	VAR robtarget Openhole_7590 := [[449.75, -1.74, 181.47], [-0.055755, 0.704905, 0.704682, -0.058508], [0,0,0,0], [9E9, 9E9, 9E9, 9E9, 9E9, 9E9]];
	VAR robtarget Openhole_7591 := [[449.26, -1.74, 181.56], [-0.057443, 0.70477, 0.704818, -0.056849], [0,0,0,0], [9E9, 9E9, 9E9, 9E9, 9E9, 9E9]];
	VAR robtarget Openhole_7592 := [[448.77, -1.75, 181.64], [-0.059082, 0.704634, 0.704954, -0.05514], [0,0,0,0], [9E9, 9E9, 9E9, 9E9, 9E9, 9E9]];
	VAR robtarget Openhole_7593 := [[448.27, -1.79, 181.72], [-0.060634, 0.704502, 0.705091, -0.053352], [0,0,0,0], [9E9, 9E9, 9E9, 9E9, 9E9, 9E9]];
	VAR robtarget Openhole_7594 := [[447.79, -1.85, 181.8], [-0.062089, 0.704376, 0.70523, -0.051487], [0,0,0,0], [9E9, 9E9, 9E9, 9E9, 9E9, 9E9]];
	VAR robtarget Openhole_7595 := [[447.3, -1.93, 181.88], [-0.063491, 0.704251, 0.705366, -0.04958], [0,0,0,0], [9E9, 9E9, 9E9, 9E9, 9E9, 9E9]];
	VAR robtarget Openhole_7596 := [[446.81, -2.01, 181.96], [-0.06485, 0.704127, 0.7055, -0.047642], [0,0,0,0], [9E9, 9E9, 9E9, 9E9, 9E9, 9E9]];
	VAR robtarget Openhole_7597 := [[445.85, -2.22, 182.11], [-0.067419, 0.703885, 0.705757, -0.043664], [0,0,0,0], [9E9, 9E9, 9E9, 9E9, 9E9, 9E9]];
	VAR robtarget Openhole_7598 := [[444.89, -2.47, 182.25], [-0.069835, 0.70365, 0.705998, -0.039588], [0,0,0,0], [9E9, 9E9, 9E9, 9E9, 9E9, 9E9]];
	VAR robtarget Openhole_7599 := [[438.19, -4.32, 183.12], [-0.086059, 0.70185, 0.707026, -0.010661], [0,0,0,0], [9E9, 9E9, 9E9, 9E9, 9E9, 9E9]];
	VAR robtarget Openhole_7600 := [[437.22, -4.54, 183.23], [-0.088535, 0.701542, 0.707076, -0.006642], [0,0,0,0], [9E9, 9E9, 9E9, 9E9, 9E9, 9E9]];
	VAR robtarget Openhole_7601 := [[431.68, -6.99, 183.59], [-0.098515, 0.700211, 0.706817, 0.020229], [0,0,0,0], [9E9, 9E9, 9E9, 9E9, 9E9, 9E9]];
	VAR robtarget Openhole_7602 := [[438.07, -6.03, 182.95], [-0.080786, 0.702477, 0.707092, -0.004576], [0,0,0,0], [9E9, 9E9, 9E9, 9E9, 9E9, 9E9]];
	VAR robtarget Openhole_7603 := [[444.39, -4.68, 182.23], [-0.064164, 0.70419, 0.706446, -0.030557], [0,0,0,0], [9E9, 9E9, 9E9, 9E9, 9E9, 9E9]];
	VAR robtarget Openhole_7604 := [[444.87, -4.57, 182.16], [-0.062897, 0.704304, 0.706356, -0.032569], [0,0,0,0], [9E9, 9E9, 9E9, 9E9, 9E9, 9E9]];
	VAR robtarget Openhole_7605 := [[445.84, -4.38, 182.04], [-0.060271, 0.704533, 0.706162, -0.036531], [0,0,0,0], [9E9, 9E9, 9E9, 9E9, 9E9, 9E9]];
	VAR robtarget Openhole_7606 := [[446.33, -4.29, 181.97], [-0.058903, 0.704649, 0.706059, -0.038474], [0,0,0,0], [9E9, 9E9, 9E9, 9E9, 9E9, 9E9]];
	VAR robtarget Openhole_7607 := [[446.82, -4.21, 181.9], [-0.057499, 0.704765, 0.705952, -0.040392], [0,0,0,0], [9E9, 9E9, 9E9, 9E9, 9E9, 9E9]];
	VAR robtarget Openhole_7608 := [[447.31, -4.15, 181.83], [-0.05605, 0.704882, 0.705842, -0.042275], [0,0,0,0], [9E9, 9E9, 9E9, 9E9, 9E9, 9E9]];
	VAR robtarget Openhole_7609 := [[447.81, -4.1, 181.76], [-0.054542, 0.705, 0.70573, -0.044111], [0,0,0,0], [9E9, 9E9, 9E9, 9E9, 9E9, 9E9]];
	VAR robtarget Openhole_7610 := [[448.3, -4.06, 181.69], [-0.053001, 0.705118, 0.705614, -0.04592], [0,0,0,0], [9E9, 9E9, 9E9, 9E9, 9E9, 9E9]];
	VAR robtarget Openhole_7611 := [[448.79, -4.06, 181.62], [-0.051319, 0.705242, 0.705503, -0.047599], [0,0,0,0], [9E9, 9E9, 9E9, 9E9, 9E9, 9E9]];
	VAR robtarget Openhole_7612 := [[449.78, -4.1, 181.48], [-0.047827, 0.705487, 0.705278, -0.050827], [0,0,0,0], [9E9, 9E9, 9E9, 9E9, 9E9, 9E9]];
	VAR robtarget Openhole_7613 := [[450.77, -4.2, 181.34], [-0.04413, 0.705728, 0.705056, -0.053821], [0,0,0,0], [9E9, 9E9, 9E9, 9E9, 9E9, 9E9]];
	VAR robtarget Openhole_7614 := [[456.16, -5.01, 180.62], [-0.022978, 0.706733, 0.703708, -0.069248], [0,0,0,0], [9E9, 9E9, 9E9, 9E9, 9E9, 9E9]];
	VAR robtarget Openhole_7615 := [[458.63, -5.19, 180.3], [-0.013888, 0.70697, 0.702918, -0.07685], [0,0,0,0], [9E9, 9E9, 9E9, 9E9, 9E9, 9E9]];
	VAR robtarget Openhole_7616 := [[459.13, -5.2, 180.24], [-0.012156, 0.707002, 0.702741, -0.078456], [0,0,0,0], [9E9, 9E9, 9E9, 9E9, 9E9, 9E9]];
	VAR robtarget Openhole_7617 := [[463.09, -5.04, 179.69], [0.000811, 0.707106, 0.701098, -0.091987], [0,0,0,0], [9E9, 9E9, 9E9, 9E9, 9E9, 9E9]];
	VAR robtarget Openhole_7618 := [[464.07, -4.96, 179.55], [0.003898, 0.707096, 0.700634, -0.095458], [0,0,0,0], [9E9, 9E9, 9E9, 9E9, 9E9, 9E9]];
	VAR robtarget Openhole_7619 := [[472.91, -4.06, 178.14], [0.030775, 0.706437, 0.695722, -0.126377], [0,0,0,0], [9E9, 9E9, 9E9, 9E9, 9E9, 9E9]];
	VAR robtarget Openhole_7620 := [[478.35, -3.86, 177.31], [0.048077, 0.705471, 0.692398, -0.143474], [0,0,0,0], [9E9, 9E9, 9E9, 9E9, 9E9, 9E9]];
	VAR robtarget Openhole_7621 := [[478.84, -3.85, 177.23], [0.04969, 0.705359, 0.692091, -0.144947], [0,0,0,0], [9E9, 9E9, 9E9, 9E9, 9E9, 9E9]];
	VAR robtarget Openhole_7622 := [[479.33, -3.86, 177.16], [0.051314, 0.705242, 0.691785, -0.146401], [0,0,0,0], [9E9, 9E9, 9E9, 9E9, 9E9, 9E9]];
	VAR robtarget Openhole_7623 := [[480.82, -3.88, 176.95], [0.056219, 0.704868, 0.690865, -0.150682], [0,0,0,0], [9E9, 9E9, 9E9, 9E9, 9E9, 9E9]];
	VAR robtarget Openhole_7624 := [[474.12, -5.49, 178.31], [0.039466, 0.706005, 0.695882, -0.125489], [0,0,0,0], [9E9, 9E9, 9E9, 9E9, 9E9, 9E9]];
	VAR robtarget Openhole_7625 := [[469.21, -6.03, 179.06], [0.024831, 0.706671, 0.698747, -0.108408], [0,0,0,0], [9E9, 9E9, 9E9, 9E9, 9E9, 9E9]];
	VAR robtarget Openhole_7626 := [[460.88, -7.27, 180.24], [0.000752, 0.707106, 0.702859, -0.077394], [0,0,0,0], [9E9, 9E9, 9E9, 9E9, 9E9, 9E9]];
	VAR robtarget Openhole_7627 := [[457.42, -7.57, 180.65], [-0.010088, 0.707035, 0.704119, -0.064938], [0,0,0,0], [9E9, 9E9, 9E9, 9E9, 9E9, 9E9]];
	VAR robtarget Openhole_7628 := [[455.43, -7.61, 180.87], [-0.016739, 0.706909, 0.704712, -0.058151], [0,0,0,0], [9E9, 9E9, 9E9, 9E9, 9E9, 9E9]];
	VAR robtarget Openhole_7629 := [[452.45, -7.48, 181.2], [-0.027374, 0.706577, 0.705437, -0.048573], [0,0,0,0], [9E9, 9E9, 9E9, 9E9, 9E9, 9E9]];
	VAR robtarget Openhole_7630 := [[448.48, -7.26, 181.64], [-0.041664, 0.705878, 0.706196, -0.035883], [0,0,0,0], [9E9, 9E9, 9E9, 9E9, 9E9, 9E9]];
	VAR robtarget Openhole_7631 := [[447.49, -7.25, 181.75], [-0.045079, 0.705668, 0.706357, -0.032546], [0,0,0,0], [9E9, 9E9, 9E9, 9E9, 9E9, 9E9]];
	VAR robtarget Openhole_7632 := [[446.49, -7.27, 181.86], [-0.048387, 0.705449, 0.706508, -0.029104], [0,0,0,0], [9E9, 9E9, 9E9, 9E9, 9E9, 9E9]];
	VAR robtarget Openhole_7633 := [[445.5, -7.33, 181.97], [-0.051524, 0.705227, 0.706647, -0.025509], [0,0,0,0], [9E9, 9E9, 9E9, 9E9, 9E9, 9E9]];
	VAR robtarget Openhole_7634 := [[444.51, -7.43, 182.08], [-0.054538, 0.705, 0.70677, -0.021812], [0,0,0,0], [9E9, 9E9, 9E9, 9E9, 9E9, 9E9]];
	VAR robtarget Openhole_7635 := [[444.02, -7.49, 182.13], [-0.056012, 0.704885, 0.706826, -0.019937], [0,0,0,0], [9E9, 9E9, 9E9, 9E9, 9E9, 9E9]];
	VAR robtarget Openhole_7636 := [[437.6, -8.31, 182.75], [-0.074742, 0.703146, 0.707092, 0.004613], [0,0,0,0], [9E9, 9E9, 9E9, 9E9, 9E9, 9E9]];
	VAR robtarget Openhole_7637 := [[423.69, -9.33, 183.94], [-0.116174, 0.697498, 0.705016, 0.054336], [0,0,0,0], [9E9, 9E9, 9E9, 9E9, 9E9, 9E9]];
	VAR robtarget Openhole_7638 := [[407.25, -10.08, 185.17], [-0.162185, 0.688256, 0.698806, 0.108027], [0,0,0,0], [9E9, 9E9, 9E9, 9E9, 9E9, 9E9]];
	VAR robtarget Openhole_7639 := [[394.36, -10.64, 185.98], [-0.19429, 0.679891, 0.691824, 0.146217], [0,0,0,0], [9E9, 9E9, 9E9, 9E9, 9E9, 9E9]];
	VAR robtarget Openhole_7640 := [[389.36, -10.64, 186.38], [-0.206348, 0.676329, 0.688912, 0.159374], [0,0,0,0], [9E9, 9E9, 9E9, 9E9, 9E9, 9E9]];
	VAR robtarget Openhole_7641 := [[362.36, -10.64, 186.47], [-0.183051, 0.683002, 0.683002, 0.183051], [0,0,0,0], [9E9, 9E9, 9E9, 9E9, 9E9, 9E9]];
	VAR robtarget Openhole_7642 := [[361.72, -33.92, 173.02], [-0.183051, 0.683002, 0.683002, 0.183051], [0,0,0,0], [9E9, 9E9, 9E9, 9E9, 9E9, 9E9]];
	VAR robtarget Openhole_7643 := [[389.32, -33.92, 172.94], [-0.14, 0.693109, 0.670339, 0.225045], [0,0,0,0], [9E9, 9E9, 9E9, 9E9, 9E9, 9E9]];
	VAR robtarget Openhole_7644 := [[399.12, -33.92, 174.34], [-0.112575, 0.698088, 0.677653, 0.201957], [0,0,0,0], [9E9, 9E9, 9E9, 9E9, 9E9, 9E9]];
	VAR robtarget Openhole_7645 := [[405.51, -35.06, 174.78], [-0.090137, 0.701338, 0.681366, 0.18905], [0,0,0,0], [9E9, 9E9, 9E9, 9E9, 9E9, 9E9]];
	VAR robtarget Openhole_7646 := [[411.91, -35.92, 175.46], [-0.067551, 0.703873, 0.685253, 0.174436], [0,0,0,0], [9E9, 9E9, 9E9, 9E9, 9E9, 9E9]];
	VAR robtarget Openhole_7647 := [[417.84, -36.39, 176.28], [-0.046962, 0.705546, 0.688953, 0.159198], [0,0,0,0], [9E9, 9E9, 9E9, 9E9, 9E9, 9E9]];
	VAR robtarget Openhole_7648 := [[421.78, -36.5, 176.91], [-0.033583, 0.706309, 0.691444, 0.148003], [0,0,0,0], [9E9, 9E9, 9E9, 9E9, 9E9, 9E9]];
	VAR robtarget Openhole_7649 := [[422.28, -36.5, 176.99], [-0.031944, 0.706385, 0.691756, 0.146538], [0,0,0,0], [9E9, 9E9, 9E9, 9E9, 9E9, 9E9]];
	VAR robtarget Openhole_7650 := [[428.18, -36.31, 178.02], [-0.012739, 0.706992, 0.69543, 0.127974], [0,0,0,0], [9E9, 9E9, 9E9, 9E9, 9E9, 9E9]];
	VAR robtarget Openhole_7651 := [[436.05, -35.81, 179.39], [0.01245, 0.706997, 0.69979, 0.101457], [0,0,0,0], [9E9, 9E9, 9E9, 9E9, 9E9, 9E9]];
	VAR robtarget Openhole_7652 := [[437.04, -35.79, 179.56], [0.015763, 0.706931, 0.700256, 0.098191], [0,0,0,0], [9E9, 9E9, 9E9, 9E9, 9E9, 9E9]];
	VAR robtarget Openhole_7653 := [[438.02, -35.8, 179.71], [0.019161, 0.706847, 0.700698, 0.094988], [0,0,0,0], [9E9, 9E9, 9E9, 9E9, 9E9, 9E9]];
	VAR robtarget Openhole_7654 := [[439.01, -35.82, 179.87], [0.022643, 0.706744, 0.701116, 0.091853], [0,0,0,0], [9E9, 9E9, 9E9, 9E9, 9E9, 9E9]];
	VAR robtarget Openhole_7655 := [[440, -35.88, 180.03], [0.026226, 0.70662, 0.701507, 0.088811], [0,0,0,0], [9E9, 9E9, 9E9, 9E9, 9E9, 9E9]];
	VAR robtarget Openhole_7656 := [[440.98, -35.98, 180.18], [0.029904, 0.706474, 0.701874, 0.085865], [0,0,0,0], [9E9, 9E9, 9E9, 9E9, 9E9, 9E9]];
	VAR robtarget Openhole_7657 := [[441.96, -36.1, 180.33], [0.033684, 0.706304, 0.702215, 0.083033], [0,0,0,0], [9E9, 9E9, 9E9, 9E9, 9E9, 9E9]];
	VAR robtarget Openhole_7658 := [[442.94, -36.26, 180.48], [0.037548, 0.706109, 0.702532, 0.080306], [0,0,0,0], [9E9, 9E9, 9E9, 9E9, 9E9, 9E9]];
	VAR robtarget Openhole_7659 := [[443.91, -36.44, 180.63], [0.041484, 0.705889, 0.702827, 0.077676], [0,0,0,0], [9E9, 9E9, 9E9, 9E9, 9E9, 9E9]];
	VAR robtarget Openhole_7660 := [[445.84, -36.87, 180.94], [0.049487, 0.705373, 0.703369, 0.072613], [0,0,0,0], [9E9, 9E9, 9E9, 9E9, 9E9, 9E9]];
	VAR robtarget Openhole_7661 := [[446.31, -37, 181.02], [0.051566, 0.705224, 0.703485, 0.071479], [0,0,0,0], [9E9, 9E9, 9E9, 9E9, 9E9, 9E9]];
	VAR robtarget Openhole_7662 := [[446.78, -37.17, 181.09], [0.053699, 0.705065, 0.703588, 0.070455], [0,0,0,0], [9E9, 9E9, 9E9, 9E9, 9E9, 9E9]];
	VAR robtarget Openhole_7663 := [[447.24, -37.35, 181.17], [0.055869, 0.704896, 0.703682, 0.069514], [0,0,0,0], [9E9, 9E9, 9E9, 9E9, 9E9, 9E9]];
	VAR robtarget Openhole_7664 := [[448.2, -37.57, 181.34], [0.059857, 0.704569, 0.703927, 0.066981], [0,0,0,0], [9E9, 9E9, 9E9, 9E9, 9E9, 9E9]];
	VAR robtarget Openhole_7665 := [[448.69, -37.57, 181.42], [0.061551, 0.704423, 0.704081, 0.065341], [0,0,0,0], [9E9, 9E9, 9E9, 9E9, 9E9, 9E9]];
	VAR robtarget Openhole_7666 := [[449.18, -37.57, 181.51], [0.063199, 0.704277, 0.704236, 0.063655], [0,0,0,0], [9E9, 9E9, 9E9, 9E9, 9E9, 9E9]];
	VAR robtarget Openhole_7667 := [[450.15, -37.36, 181.68], [0.065802, 0.704038, 0.70458, 0.059727], [0,0,0,0], [9E9, 9E9, 9E9, 9E9, 9E9, 9E9]];
	VAR robtarget Openhole_7668 := [[450.62, -37.23, 181.76], [0.066984, 0.703927, 0.70475, 0.057688], [0,0,0,0], [9E9, 9E9, 9E9, 9E9, 9E9, 9E9]];
	VAR robtarget Openhole_7669 := [[451.1, -37.12, 181.85], [0.068226, 0.703808, 0.704911, 0.055684], [0,0,0,0], [9E9, 9E9, 9E9, 9E9, 9E9, 9E9]];
	VAR robtarget Openhole_7670 := [[451.58, -36.98, 181.93], [0.069387, 0.703694, 0.70507, 0.053631], [0,0,0,0], [9E9, 9E9, 9E9, 9E9, 9E9, 9E9]];
	VAR robtarget Openhole_7671 := [[459.65, -34.59, 183.08], [0.088452, 0.701553, 0.706872, 0.018235], [0,0,0,0], [9E9, 9E9, 9E9, 9E9, 9E9, 9E9]];
	VAR robtarget Openhole_7672 := [[460.13, -34.45, 183.14], [0.089592, 0.701408, 0.706922, 0.016165], [0,0,0,0], [9E9, 9E9, 9E9, 9E9, 9E9, 9E9]];
	VAR robtarget Openhole_7673 := [[461.11, -32.96, 183.12], [0.087897, 0.701622, 0.707063, 0.007883], [0,0,0,0], [9E9, 9E9, 9E9, 9E9, 9E9, 9E9]];
	VAR robtarget Openhole_7674 := [[460.14, -33.18, 183.01], [0.085435, 0.701927, 0.707006, 0.011915], [0,0,0,0], [9E9, 9E9, 9E9, 9E9, 9E9, 9E9]];
	VAR robtarget Openhole_7675 := [[453.43, -34.99, 182.17], [0.069075, 0.703725, 0.70593, 0.040779], [0,0,0,0], [9E9, 9E9, 9E9, 9E9, 9E9, 9E9]];
	VAR robtarget Openhole_7676 := [[452.47, -35.23, 182.03], [0.066594, 0.703964, 0.705685, 0.044816], [0,0,0,0], [9E9, 9E9, 9E9, 9E9, 9E9, 9E9]];
	VAR robtarget Openhole_7677 := [[451.98, -35.33, 181.96], [0.065304, 0.704085, 0.705556, 0.046802], [0,0,0,0], [9E9, 9E9, 9E9, 9E9, 9E9, 9E9]];
	VAR robtarget Openhole_7678 := [[451.5, -35.42, 181.88], [0.063974, 0.704207, 0.705424, 0.04876], [0,0,0,0], [9E9, 9E9, 9E9, 9E9, 9E9, 9E9]];
	VAR robtarget Openhole_7679 := [[451.01, -35.49, 181.8], [0.062545, 0.704335, 0.705291, 0.050648], [0,0,0,0], [9E9, 9E9, 9E9, 9E9, 9E9, 9E9]];
	VAR robtarget Openhole_7680 := [[450.52, -35.55, 181.73], [0.06107, 0.704465, 0.705155, 0.052498], [0,0,0,0], [9E9, 9E9, 9E9, 9E9, 9E9, 9E9]];
	VAR robtarget Openhole_7681 := [[450.03, -35.58, 181.65], [0.059515, 0.704598, 0.70502, 0.054283], [0,0,0,0], [9E9, 9E9, 9E9, 9E9, 9E9, 9E9]];
	VAR robtarget Openhole_7682 := [[449.53, -35.6, 181.57], [0.057897, 0.704733, 0.704885, 0.056013], [0,0,0,0], [9E9, 9E9, 9E9, 9E9, 9E9, 9E9]];
	VAR robtarget Openhole_7683 := [[449.04, -35.59, 181.49], [0.056177, 0.704872, 0.704754, 0.05764], [0,0,0,0], [9E9, 9E9, 9E9, 9E9, 9E9, 9E9]];
	VAR robtarget Openhole_7684 := [[448.55, -35.55, 181.41], [0.05438, 0.705013, 0.704626, 0.059182], [0,0,0,0], [9E9, 9E9, 9E9, 9E9, 9E9, 9E9]];
	VAR robtarget Openhole_7685 := [[448.06, -35.5, 181.34], [0.052527, 0.705153, 0.7045, 0.06066], [0,0,0,0], [9E9, 9E9, 9E9, 9E9, 9E9, 9E9]];
	VAR robtarget Openhole_7686 := [[447.57, -35.43, 181.26], [0.050625, 0.705292, 0.704377, 0.062073], [0,0,0,0], [9E9, 9E9, 9E9, 9E9, 9E9, 9E9]];
	VAR robtarget Openhole_7687 := [[446.59, -35.25, 181.11], [0.04671, 0.705562, 0.704136, 0.064752], [0,0,0,0], [9E9, 9E9, 9E9, 9E9, 9E9, 9E9]];
	VAR robtarget Openhole_7688 := [[443.68, -34.65, 180.69], [0.034788, 0.706251, 0.703375, 0.072552], [0,0,0,0], [9E9, 9E9, 9E9, 9E9, 9E9, 9E9]];
	VAR robtarget Openhole_7689 := [[441.73, -34.35, 180.42], [0.027076, 0.706588, 0.702783, 0.078074], [0,0,0,0], [9E9, 9E9, 9E9, 9E9, 9E9, 9E9]];
	VAR robtarget Openhole_7690 := [[440.74, -34.25, 180.28], [0.023353, 0.706721, 0.702453, 0.080994], [0,0,0,0], [9E9, 9E9, 9E9, 9E9, 9E9, 9E9]];
	VAR robtarget Openhole_7691 := [[439.75, -34.17, 180.14], [0.019722, 0.706832, 0.702098, 0.084012], [0,0,0,0], [9E9, 9E9, 9E9, 9E9, 9E9, 9E9]];
	VAR robtarget Openhole_7692 := [[438.76, -34.13, 180], [0.016187, 0.706921, 0.701719, 0.087122], [0,0,0,0], [9E9, 9E9, 9E9, 9E9, 9E9, 9E9]];
	VAR robtarget Openhole_7693 := [[437.77, -34.12, 179.86], [0.012758, 0.706992, 0.701314, 0.090326], [0,0,0,0], [9E9, 9E9, 9E9, 9E9, 9E9, 9E9]];
	VAR robtarget Openhole_7694 := [[437.28, -34.12, 179.79], [0.01108, 0.70702, 0.701102, 0.091956], [0,0,0,0], [9E9, 9E9, 9E9, 9E9, 9E9, 9E9]];
	VAR robtarget Openhole_7695 := [[431.85, -34.44, 178.95], [-0.00638, 0.707078, 0.698424, 0.110474], [0,0,0,0], [9E9, 9E9, 9E9, 9E9, 9E9, 9E9]];
	VAR robtarget Openhole_7696 := [[424.96, -34.89, 177.82], [-0.028192, 0.706545, 0.694415, 0.133373], [0,0,0,0], [9E9, 9E9, 9E9, 9E9, 9E9, 9E9]];
	VAR robtarget Openhole_7697 := [[422, -34.94, 177.35], [-0.037884, 0.706091, 0.692603, 0.142482], [0,0,0,0], [9E9, 9E9, 9E9, 9E9, 9E9, 9E9]];
	VAR robtarget Openhole_7698 := [[421.5, -34.94, 177.28], [-0.039531, 0.706001, 0.6923, 0.143945], [0,0,0,0], [9E9, 9E9, 9E9, 9E9, 9E9, 9E9]];
	VAR robtarget Openhole_7699 := [[415.57, -34.71, 176.45], [-0.059667, 0.704585, 0.688649, 0.160508], [0,0,0,0], [9E9, 9E9, 9E9, 9E9, 9E9, 9E9]];
	VAR robtarget Openhole_7700 := [[409.14, -34.09, 175.71], [-0.081938, 0.702343, 0.684724, 0.176502], [0,0,0,0], [9E9, 9E9, 9E9, 9E9, 9E9, 9E9]];
	VAR robtarget Openhole_7701 := [[404.2, -33.45, 175.28], [-0.099015, 0.70014, 0.681745, 0.187681], [0,0,0,0], [9E9, 9E9, 9E9, 9E9, 9E9, 9E9]];
	VAR robtarget Openhole_7702 := [[411.67, -32.92, 176.51], [-0.077704, 0.702824, 0.687349, 0.165988], [0,0,0,0], [9E9, 9E9, 9E9, 9E9, 9E9, 9E9]];
	VAR robtarget Openhole_7703 := [[418.12, -33.28, 177.26], [-0.055972, 0.704888, 0.691289, 0.148726], [0,0,0,0], [9E9, 9E9, 9E9, 9E9, 9E9, 9E9]];
	VAR robtarget Openhole_7704 := [[420.6, -33.32, 177.59], [-0.047766, 0.705492, 0.692797, 0.141538], [0,0,0,0], [9E9, 9E9, 9E9, 9E9, 9E9, 9E9]];
	VAR robtarget Openhole_7705 := [[421.09, -33.31, 177.66], [-0.046147, 0.705599, 0.693098, 0.140056], [0,0,0,0], [9E9, 9E9, 9E9, 9E9, 9E9, 9E9]];
	VAR robtarget Openhole_7706 := [[426.53, -33.08, 178.46], [-0.028845, 0.706518, 0.696362, 0.122803], [0,0,0,0], [9E9, 9E9, 9E9, 9E9, 9E9, 9E9]];
	VAR robtarget Openhole_7707 := [[436.37, -32.09, 179.91], [0.001199, 0.707106, 0.701578, 0.088254], [0,0,0,0], [9E9, 9E9, 9E9, 9E9, 9E9, 9E9]];
	VAR robtarget Openhole_7708 := [[438.85, -31.99, 180.23], [0.009317, 0.707045, 0.70259, 0.079793], [0,0,0,0], [9E9, 9E9, 9E9, 9E9, 9E9, 9E9]];
	VAR robtarget Openhole_7709 := [[439.84, -31.99, 180.36], [0.012734, 0.706992, 0.702952, 0.07654], [0,0,0,0], [9E9, 9E9, 9E9, 9E9, 9E9, 9E9]];
	VAR robtarget Openhole_7710 := [[441.33, -32.04, 180.54], [0.017999, 0.706878, 0.703454, 0.071779], [0,0,0,0], [9E9, 9E9, 9E9, 9E9, 9E9, 9E9]];
	VAR robtarget Openhole_7711 := [[442.32, -32.11, 180.66], [0.021607, 0.706777, 0.703762, 0.068696], [0,0,0,0], [9E9, 9E9, 9E9, 9E9, 9E9, 9E9]];
	VAR robtarget Openhole_7712 := [[442.81, -32.16, 180.72], [0.023462, 0.706717, 0.703905, 0.06721], [0,0,0,0], [9E9, 9E9, 9E9, 9E9, 9E9, 9E9]];
	VAR robtarget Openhole_7713 := [[447.23, -32.82, 181.26], [0.040783, 0.70593, 0.704996, 0.054591], [0,0,0,0], [9E9, 9E9, 9E9, 9E9, 9E9, 9E9]];
	VAR robtarget Openhole_7714 := [[448.21, -32.96, 181.39], [0.044601, 0.705699, 0.705211, 0.051745], [0,0,0,0], [9E9, 9E9, 9E9, 9E9, 9E9, 9E9]];
	VAR robtarget Openhole_7715 := [[448.7, -33.01, 181.45], [0.046456, 0.705579, 0.705319, 0.050252], [0,0,0,0], [9E9, 9E9, 9E9, 9E9, 9E9, 9E9]];
	VAR robtarget Openhole_7716 := [[449.2, -33.05, 181.52], [0.048263, 0.705458, 0.705427, 0.048706], [0,0,0,0], [9E9, 9E9, 9E9, 9E9, 9E9, 9E9]];
	VAR robtarget Openhole_7717 := [[449.69, -33.07, 181.59], [0.05002, 0.705335, 0.705536, 0.047102], [0,0,0,0], [9E9, 9E9, 9E9, 9E9, 9E9, 9E9]];
	VAR robtarget Openhole_7718 := [[450.19, -33.08, 181.65], [0.051725, 0.705212, 0.705645, 0.045443], [0,0,0,0], [9E9, 9E9, 9E9, 9E9, 9E9, 9E9]];
	VAR robtarget Openhole_7719 := [[451.18, -33.03, 181.79], [0.054938, 0.704969, 0.705862, 0.041938], [0,0,0,0], [9E9, 9E9, 9E9, 9E9, 9E9, 9E9]];
	VAR robtarget Openhole_7720 := [[451.67, -32.99, 181.85], [0.056457, 0.704849, 0.705968, 0.04011], [0,0,0,0], [9E9, 9E9, 9E9, 9E9, 9E9, 9E9]];
	VAR robtarget Openhole_7721 := [[452.16, -32.92, 181.92], [0.057903, 0.704732, 0.706073, 0.038223], [0,0,0,0], [9E9, 9E9, 9E9, 9E9, 9E9, 9E9]];
	VAR robtarget Openhole_7722 := [[452.65, -32.84, 181.98], [0.059299, 0.704616, 0.706174, 0.036299], [0,0,0,0], [9E9, 9E9, 9E9, 9E9, 9E9, 9E9]];
	VAR robtarget Openhole_7723 := [[453.63, -32.66, 182.1], [0.061962, 0.704387, 0.706366, 0.032359], [0,0,0,0], [9E9, 9E9, 9E9, 9E9, 9E9, 9E9]];
	VAR robtarget Openhole_7724 := [[460.44, -31.22, 182.84], [0.07991, 0.702577, 0.707093, 0.004382], [0,0,0,0], [9E9, 9E9, 9E9, 9E9, 9E9, 9E9]];
	VAR robtarget Openhole_7725 := [[466.84, -30.31, 183.44], [0.097818, 0.700308, 0.706815, -0.020309], [0,0,0,0], [9E9, 9E9, 9E9, 9E9, 9E9, 9E9]];
	VAR robtarget Openhole_7726 := [[476.26, -29.36, 184.22], [0.12433, 0.69609, 0.704993, -0.054634], [0,0,0,0], [9E9, 9E9, 9E9, 9E9, 9E9, 9E9]];
	VAR robtarget Openhole_7727 := [[470.3, -26.56, 183.06], [0.096566, 0.700482, 0.705722, -0.044238], [0,0,0,0], [9E9, 9E9, 9E9, 9E9, 9E9, 9E9]];
	VAR robtarget Openhole_7728 := [[465.31, -26.64, 182.71], [0.080722, 0.702484, 0.706578, -0.027351], [0,0,0,0], [9E9, 9E9, 9E9, 9E9, 9E9, 9E9]];
	VAR robtarget Openhole_7729 := [[464.82, -26.64, 182.67], [0.079088, 0.70267, 0.70664, -0.025682], [0,0,0,0], [9E9, 9E9, 9E9, 9E9, 9E9, 9E9]];
	VAR robtarget Openhole_7730 := [[463.82, -26.63, 182.6], [0.075801, 0.703032, 0.706754, -0.022343], [0,0,0,0], [9E9, 9E9, 9E9, 9E9, 9E9, 9E9]];
	VAR robtarget Openhole_7731 := [[463.32, -26.64, 182.56], [0.074164, 0.703207, 0.706805, -0.020661], [0,0,0,0], [9E9, 9E9, 9E9, 9E9, 9E9, 9E9]];
	VAR robtarget Openhole_7732 := [[462.82, -26.63, 182.53], [0.072502, 0.70338, 0.706852, -0.018998], [0,0,0,0], [9E9, 9E9, 9E9, 9E9, 9E9, 9E9]];
	VAR robtarget Openhole_7733 := [[459.33, -26.59, 182.27], [0.060784, 0.704489, 0.707069, -0.007327], [0,0,0,0], [9E9, 9E9, 9E9, 9E9, 9E9, 9E9]];
	VAR robtarget Openhole_7734 := [[458.83, -26.59, 182.23], [0.059117, 0.704631, 0.707084, -0.005637], [0,0,0,0], [9E9, 9E9, 9E9, 9E9, 9E9, 9E9]];
	VAR robtarget Openhole_7735 := [[458.33, -26.6, 182.2], [0.057459, 0.704768, 0.707096, -0.003935], [0,0,0,0], [9E9, 9E9, 9E9, 9E9, 9E9, 9E9]];
	VAR robtarget Openhole_7736 := [[457.83, -26.59, 182.16], [0.055777, 0.704903, 0.707103, -0.002253], [0,0,0,0], [9E9, 9E9, 9E9, 9E9, 9E9, 9E9]];
	VAR robtarget Openhole_7737 := [[456.34, -26.58, 182.05], [0.050691, 0.705287, 0.707101, 0.002767], [0,0,0,0], [9E9, 9E9, 9E9, 9E9, 9E9, 9E9]];
	VAR robtarget Openhole_7738 := [[455.34, -26.54, 181.97], [0.04721, 0.705529, 0.707081, 0.006033], [0,0,0,0], [9E9, 9E9, 9E9, 9E9, 9E9, 9E9]];
	VAR robtarget Openhole_7739 := [[454.85, -26.49, 181.94], [0.045376, 0.705649, 0.707066, 0.007562], [0,0,0,0], [9E9, 9E9, 9E9, 9E9, 9E9, 9E9]];
	VAR robtarget Openhole_7740 := [[454.35, -26.44, 181.9], [0.043506, 0.705767, 0.707049, 0.009049], [0,0,0,0], [9E9, 9E9, 9E9, 9E9, 9E9, 9E9]];
	VAR robtarget Openhole_7741 := [[453.86, -26.35, 181.86], [0.041562, 0.705884, 0.70703, 0.01044], [0,0,0,0], [9E9, 9E9, 9E9, 9E9, 9E9, 9E9]];
	VAR robtarget Openhole_7742 := [[453.37, -26.25, 181.82], [0.03957, 0.705999, 0.707009, 0.011766], [0,0,0,0], [9E9, 9E9, 9E9, 9E9, 9E9, 9E9]];
	VAR robtarget Openhole_7743 := [[452.79, -25.92, 181.77], [0.036472, 0.706166, 0.706994, 0.012621], [0,0,0,0], [9E9, 9E9, 9E9, 9E9, 9E9, 9E9]];
	VAR robtarget Openhole_7744 := [[454.94, -24.42, 181.83], [0.038676, 0.706048, 0.707107, 0.000228], [0,0,0,0], [9E9, 9E9, 9E9, 9E9, 9E9, 9E9]];
	VAR robtarget Openhole_7745 := [[455.54, -24.57, 181.87], [0.041225, 0.705904, 0.707106, -0.001297], [0,0,0,0], [9E9, 9E9, 9E9, 9E9, 9E9, 9E9]];
	VAR robtarget Openhole_7746 := [[456.54, -24.66, 181.93], [0.044874, 0.705681, 0.707093, -0.004383], [0,0,0,0], [9E9, 9E9, 9E9, 9E9, 9E9, 9E9]];
	VAR robtarget Openhole_7747 := [[457.04, -24.68, 181.96], [0.046645, 0.705567, 0.707081, -0.005982], [0,0,0,0], [9E9, 9E9, 9E9, 9E9, 9E9, 9E9]];
	VAR robtarget Openhole_7748 := [[460.52, -24.98, 182.18], [0.059311, 0.704615, 0.706908, -0.016769], [0,0,0,0], [9E9, 9E9, 9E9, 9E9, 9E9, 9E9]];
	VAR robtarget Openhole_7749 := [[457.19, -28.45, 182.25], [0.059837, 0.70457, 0.70708, 0.006176], [0,0,0,0], [9E9, 9E9, 9E9, 9E9, 9E9, 9E9]];
	VAR robtarget Openhole_7750 := [[454.2, -28.65, 181.99], [0.050478, 0.705303, 0.706903, 0.01699], [0,0,0,0], [9E9, 9E9, 9E9, 9E9, 9E9, 9E9]];
	VAR robtarget Openhole_7751 := [[453.71, -28.66, 181.95], [0.048836, 0.705418, 0.706859, 0.018724], [0,0,0,0], [9E9, 9E9, 9E9, 9E9, 9E9, 9E9]];
	VAR robtarget Openhole_7752 := [[452.71, -28.67, 181.85], [0.045488, 0.705642, 0.70676, 0.022133], [0,0,0,0], [9E9, 9E9, 9E9, 9E9, 9E9, 9E9]];
	VAR robtarget Openhole_7753 := [[449.23, -28.52, 181.53], [0.033165, 0.706329, 0.706314, 0.033467], [0,0,0,0], [9E9, 9E9, 9E9, 9E9, 9E9, 9E9]];
	VAR robtarget Openhole_7754 := [[448.73, -28.52, 181.49], [0.031442, 0.706407, 0.706234, 0.035127], [0,0,0,0], [9E9, 9E9, 9E9, 9E9, 9E9, 9E9]];
	VAR robtarget Openhole_7755 := [[448.23, -28.52, 181.44], [0.029744, 0.706481, 0.706148, 0.036814], [0,0,0,0], [9E9, 9E9, 9E9, 9E9, 9E9, 9E9]];
	VAR robtarget Openhole_7756 := [[447.24, -28.52, 181.35], [0.026357, 0.706615, 0.705964, 0.040193], [0,0,0,0], [9E9, 9E9, 9E9, 9E9, 9E9, 9E9]];
	VAR robtarget Openhole_7757 := [[444.75, -28.61, 181.12], [0.01815, 0.706874, 0.705416, 0.048872], [0,0,0,0], [9E9, 9E9, 9E9, 9E9, 9E9, 9E9]];
	VAR robtarget Openhole_7758 := [[443.26, -28.67, 180.98], [0.013272, 0.706982, 0.705034, 0.054102], [0,0,0,0], [9E9, 9E9, 9E9, 9E9, 9E9, 9E9]];
	VAR robtarget Openhole_7759 := [[444.55, -31.6, 180.96], [0.02758, 0.706569, 0.704595, 0.059544], [0,0,0,0], [9E9, 9E9, 9E9, 9E9, 9E9, 9E9]];
	VAR robtarget Openhole_7760 := [[445.54, -31.73, 181.08], [0.03138, 0.70641, 0.704833, 0.056663], [0,0,0,0], [9E9, 9E9, 9E9, 9E9, 9E9, 9E9]];
	VAR robtarget Openhole_7761 := [[446.52, -31.9, 181.19], [0.035276, 0.706226, 0.705049, 0.05391], [0,0,0,0], [9E9, 9E9, 9E9, 9E9, 9E9, 9E9]];
	VAR robtarget Openhole_7762 := [[448.49, -32.14, 181.43], [0.042816, 0.705809, 0.705471, 0.048074], [0,0,0,0], [9E9, 9E9, 9E9, 9E9, 9E9, 9E9]];
	VAR robtarget Openhole_7763 := [[448.98, -32.18, 181.5], [0.044643, 0.705696, 0.705573, 0.046543], [0,0,0,0], [9E9, 9E9, 9E9, 9E9, 9E9, 9E9]];
	VAR robtarget Openhole_7764 := [[449.48, -32.21, 181.56], [0.046426, 0.705581, 0.705676, 0.044962], [0,0,0,0], [9E9, 9E9, 9E9, 9E9, 9E9, 9E9]];
	VAR robtarget Openhole_7765 := [[449.97, -32.23, 181.62], [0.048173, 0.705464, 0.705777, 0.043345], [0,0,0,0], [9E9, 9E9, 9E9, 9E9, 9E9, 9E9]];
	VAR robtarget Openhole_7766 := [[450.47, -32.23, 181.68], [0.049855, 0.705347, 0.705879, 0.041659], [0,0,0,0], [9E9, 9E9, 9E9, 9E9, 9E9, 9E9]];
	VAR robtarget Openhole_7767 := [[450.97, -32.22, 181.75], [0.051492, 0.705229, 0.705978, 0.039931], [0,0,0,0], [9E9, 9E9, 9E9, 9E9, 9E9, 9E9]];
	VAR robtarget Openhole_7768 := [[451.46, -32.18, 181.81], [0.053057, 0.705113, 0.706078, 0.038137], [0,0,0,0], [9E9, 9E9, 9E9, 9E9, 9E9, 9E9]];
	VAR robtarget Openhole_7769 := [[451.96, -32.13, 181.87], [0.054571, 0.704998, 0.706174, 0.036302], [0,0,0,0], [9E9, 9E9, 9E9, 9E9, 9E9, 9E9]];
	VAR robtarget Openhole_7770 := [[452.45, -32.07, 181.93], [0.056024, 0.704884, 0.706269, 0.034416], [0,0,0,0], [9E9, 9E9, 9E9, 9E9, 9E9, 9E9]];
	VAR robtarget Openhole_7771 := [[453.43, -31.9, 182.05], [0.058774, 0.70466, 0.706447, 0.03053], [0,0,0,0], [9E9, 9E9, 9E9, 9E9, 9E9, 9E9]];
	VAR robtarget Openhole_7772 := [[452.74, -30.49, 181.92], [0.051737, 0.705211, 0.706546, 0.028148], [0,0,0,0], [9E9, 9E9, 9E9, 9E9, 9E9, 9E9]];
	VAR robtarget Openhole_7773 := [[451.25, -30.57, 181.75], [0.046945, 0.705547, 0.706315, 0.033461], [0,0,0,0], [9E9, 9E9, 9E9, 9E9, 9E9, 9E9]];
	VAR robtarget Openhole_7774 := [[450.76, -30.57, 181.7], [0.045265, 0.705656, 0.706232, 0.035156], [0,0,0,0], [9E9, 9E9, 9E9, 9E9, 9E9, 9E9]];
	VAR robtarget Openhole_7775 := [[450.26, -30.57, 181.64], [0.043559, 0.705764, 0.706147, 0.036824], [0,0,0,0], [9E9, 9E9, 9E9, 9E9, 9E9, 9E9]];
	VAR robtarget Openhole_7776 := [[446.79, -30.31, 181.26], [0.030887, 0.706432, 0.705495, 0.047722], [0,0,0,0], [9E9, 9E9, 9E9, 9E9, 9E9, 9E9]];

	PROC MainOpenhole()
		moveJ Openhole_0, v10, fine, pHeader\WObj:=wobj0;
		MoveL Openhole_1, v10, fine, pHeader\WObj:=wobj0;
		MoveL Openhole_2, v10, fine, pHeader\WObj:=wobj0;
		MoveL Openhole_3, v10, fine, pHeader\WObj:=wobj0;
		MoveL Openhole_4, v10, fine, pHeader\WObj:=wobj0;
		MoveL Openhole_5, v10, fine, pHeader\WObj:=wobj0;
		MoveL Openhole_6, v10, fine, pHeader\WObj:=wobj0;
		MoveL Openhole_7, v10, fine, pHeader\WObj:=wobj0;
		MoveL Openhole_8, v10, fine, pHeader\WObj:=wobj0;
		MoveL Openhole_9, v10, fine, pHeader\WObj:=wobj0;
		MoveL Openhole_10, v10, fine, pHeader\WObj:=wobj0;
		MoveL Openhole_11, v10, fine, pHeader\WObj:=wobj0;
		MoveL Openhole_12, v10, fine, pHeader\WObj:=wobj0;
		MoveL Openhole_13, v10, fine, pHeader\WObj:=wobj0;
		MoveL Openhole_14, v10, fine, pHeader\WObj:=wobj0;
		MoveL Openhole_15, v10, fine, pHeader\WObj:=wobj0;
		MoveL Openhole_16, v10, fine, pHeader\WObj:=wobj0;
		MoveL Openhole_17, v10, fine, pHeader\WObj:=wobj0;
		MoveL Openhole_18, v10, fine, pHeader\WObj:=wobj0;
		MoveL Openhole_19, v10, fine, pHeader\WObj:=wobj0;
		MoveL Openhole_20, v10, fine, pHeader\WObj:=wobj0;
		MoveL Openhole_21, v10, fine, pHeader\WObj:=wobj0;
		MoveL Openhole_22, v10, fine, pHeader\WObj:=wobj0;
		MoveL Openhole_23, v10, fine, pHeader\WObj:=wobj0;
		MoveL Openhole_24, v10, fine, pHeader\WObj:=wobj0;
		MoveL Openhole_25, v10, fine, pHeader\WObj:=wobj0;
		MoveL Openhole_26, v10, fine, pHeader\WObj:=wobj0;
		MoveL Openhole_27, v10, fine, pHeader\WObj:=wobj0;
		MoveL Openhole_28, v10, fine, pHeader\WObj:=wobj0;
		MoveL Openhole_29, v10, fine, pHeader\WObj:=wobj0;
		MoveL Openhole_30, v10, fine, pHeader\WObj:=wobj0;
		MoveL Openhole_31, v10, fine, pHeader\WObj:=wobj0;
		MoveL Openhole_32, v10, fine, pHeader\WObj:=wobj0;
		MoveL Openhole_33, v10, fine, pHeader\WObj:=wobj0;
		MoveL Openhole_34, v10, fine, pHeader\WObj:=wobj0;
		MoveL Openhole_35, v10, fine, pHeader\WObj:=wobj0;
		MoveL Openhole_36, v10, fine, pHeader\WObj:=wobj0;
		MoveL Openhole_37, v10, fine, pHeader\WObj:=wobj0;
		MoveL Openhole_38, v10, fine, pHeader\WObj:=wobj0;
		MoveL Openhole_39, v10, fine, pHeader\WObj:=wobj0;
		MoveL Openhole_40, v10, fine, pHeader\WObj:=wobj0;
		MoveL Openhole_41, v10, fine, pHeader\WObj:=wobj0;
		MoveL Openhole_42, v10, fine, pHeader\WObj:=wobj0;
		MoveL Openhole_43, v10, fine, pHeader\WObj:=wobj0;
		MoveL Openhole_44, v10, fine, pHeader\WObj:=wobj0;
		MoveL Openhole_45, v10, fine, pHeader\WObj:=wobj0;
		MoveL Openhole_46, v10, fine, pHeader\WObj:=wobj0;
		MoveL Openhole_47, v10, fine, pHeader\WObj:=wobj0;
		MoveL Openhole_48, v10, fine, pHeader\WObj:=wobj0;
		MoveL Openhole_49, v10, fine, pHeader\WObj:=wobj0;
		MoveL Openhole_50, v10, fine, pHeader\WObj:=wobj0;
		MoveL Openhole_51, v10, fine, pHeader\WObj:=wobj0;
		MoveL Openhole_52, v10, fine, pHeader\WObj:=wobj0;
		MoveL Openhole_53, v10, fine, pHeader\WObj:=wobj0;
		MoveL Openhole_54, v10, fine, pHeader\WObj:=wobj0;
		MoveL Openhole_55, v10, fine, pHeader\WObj:=wobj0;
		MoveL Openhole_56, v10, fine, pHeader\WObj:=wobj0;
		MoveL Openhole_57, v10, fine, pHeader\WObj:=wobj0;
		MoveL Openhole_58, v10, fine, pHeader\WObj:=wobj0;
		MoveL Openhole_59, v10, fine, pHeader\WObj:=wobj0;
		MoveL Openhole_60, v10, fine, pHeader\WObj:=wobj0;
		MoveL Openhole_61, v10, fine, pHeader\WObj:=wobj0;
		MoveL Openhole_62, v10, fine, pHeader\WObj:=wobj0;
		MoveL Openhole_63, v10, fine, pHeader\WObj:=wobj0;
		MoveL Openhole_64, v10, fine, pHeader\WObj:=wobj0;
		MoveL Openhole_65, v10, fine, pHeader\WObj:=wobj0;
		MoveL Openhole_66, v10, fine, pHeader\WObj:=wobj0;
		MoveL Openhole_67, v10, fine, pHeader\WObj:=wobj0;
		MoveL Openhole_68, v10, fine, pHeader\WObj:=wobj0;
		MoveL Openhole_69, v10, fine, pHeader\WObj:=wobj0;
		MoveL Openhole_70, v10, fine, pHeader\WObj:=wobj0;
		MoveL Openhole_71, v10, fine, pHeader\WObj:=wobj0;
		MoveL Openhole_72, v10, fine, pHeader\WObj:=wobj0;
		MoveL Openhole_73, v10, fine, pHeader\WObj:=wobj0;
		MoveL Openhole_74, v10, fine, pHeader\WObj:=wobj0;
		MoveL Openhole_75, v10, fine, pHeader\WObj:=wobj0;
		MoveL Openhole_76, v10, fine, pHeader\WObj:=wobj0;
		MoveL Openhole_77, v10, fine, pHeader\WObj:=wobj0;
		MoveL Openhole_78, v10, fine, pHeader\WObj:=wobj0;
		MoveL Openhole_79, v10, fine, pHeader\WObj:=wobj0;
		MoveL Openhole_80, v10, fine, pHeader\WObj:=wobj0;
		MoveL Openhole_81, v10, fine, pHeader\WObj:=wobj0;
		MoveL Openhole_82, v10, fine, pHeader\WObj:=wobj0;
		MoveL Openhole_83, v10, fine, pHeader\WObj:=wobj0;
		MoveL Openhole_84, v10, fine, pHeader\WObj:=wobj0;
		MoveL Openhole_85, v10, fine, pHeader\WObj:=wobj0;
		MoveL Openhole_86, v10, fine, pHeader\WObj:=wobj0;
		MoveL Openhole_87, v10, fine, pHeader\WObj:=wobj0;
		MoveL Openhole_88, v10, fine, pHeader\WObj:=wobj0;
		MoveL Openhole_89, v10, fine, pHeader\WObj:=wobj0;
		MoveL Openhole_90, v10, fine, pHeader\WObj:=wobj0;
		MoveL Openhole_91, v10, fine, pHeader\WObj:=wobj0;
		MoveL Openhole_92, v10, fine, pHeader\WObj:=wobj0;
		MoveL Openhole_93, v10, fine, pHeader\WObj:=wobj0;
		MoveL Openhole_94, v10, fine, pHeader\WObj:=wobj0;
		MoveL Openhole_95, v10, fine, pHeader\WObj:=wobj0;
		MoveL Openhole_96, v10, fine, pHeader\WObj:=wobj0;
		MoveL Openhole_97, v10, fine, pHeader\WObj:=wobj0;
		MoveL Openhole_98, v10, fine, pHeader\WObj:=wobj0;
		MoveL Openhole_99, v10, fine, pHeader\WObj:=wobj0;
		MoveL Openhole_100, v10, fine, pHeader\WObj:=wobj0;
		MoveL Openhole_101, v10, fine, pHeader\WObj:=wobj0;
		MoveL Openhole_102, v10, fine, pHeader\WObj:=wobj0;
		MoveL Openhole_103, v10, fine, pHeader\WObj:=wobj0;
		MoveL Openhole_104, v10, fine, pHeader\WObj:=wobj0;
		MoveL Openhole_105, v10, fine, pHeader\WObj:=wobj0;
		MoveL Openhole_106, v10, fine, pHeader\WObj:=wobj0;
		MoveL Openhole_107, v10, fine, pHeader\WObj:=wobj0;
		MoveL Openhole_108, v10, fine, pHeader\WObj:=wobj0;
		MoveL Openhole_109, v10, fine, pHeader\WObj:=wobj0;
		MoveL Openhole_110, v10, fine, pHeader\WObj:=wobj0;
		MoveL Openhole_111, v10, fine, pHeader\WObj:=wobj0;
		MoveL Openhole_112, v10, fine, pHeader\WObj:=wobj0;
		MoveL Openhole_113, v10, fine, pHeader\WObj:=wobj0;
		MoveL Openhole_114, v10, fine, pHeader\WObj:=wobj0;
		MoveL Openhole_115, v10, fine, pHeader\WObj:=wobj0;
		MoveL Openhole_116, v10, fine, pHeader\WObj:=wobj0;
		MoveL Openhole_117, v10, fine, pHeader\WObj:=wobj0;
		MoveL Openhole_118, v10, fine, pHeader\WObj:=wobj0;
		MoveL Openhole_119, v10, fine, pHeader\WObj:=wobj0;
		MoveL Openhole_120, v10, fine, pHeader\WObj:=wobj0;
		MoveL Openhole_121, v10, fine, pHeader\WObj:=wobj0;
		MoveL Openhole_122, v10, fine, pHeader\WObj:=wobj0;
		MoveL Openhole_123, v10, fine, pHeader\WObj:=wobj0;
		MoveL Openhole_124, v10, fine, pHeader\WObj:=wobj0;
		MoveL Openhole_125, v10, fine, pHeader\WObj:=wobj0;
		MoveL Openhole_126, v10, fine, pHeader\WObj:=wobj0;
		MoveL Openhole_127, v10, fine, pHeader\WObj:=wobj0;
		MoveL Openhole_128, v10, fine, pHeader\WObj:=wobj0;
		MoveL Openhole_129, v10, fine, pHeader\WObj:=wobj0;
		MoveL Openhole_130, v10, fine, pHeader\WObj:=wobj0;
		MoveL Openhole_131, v10, fine, pHeader\WObj:=wobj0;
		MoveL Openhole_132, v10, fine, pHeader\WObj:=wobj0;
		MoveL Openhole_133, v10, fine, pHeader\WObj:=wobj0;
		MoveL Openhole_134, v10, fine, pHeader\WObj:=wobj0;
		MoveL Openhole_135, v10, fine, pHeader\WObj:=wobj0;
		MoveL Openhole_136, v10, fine, pHeader\WObj:=wobj0;
		MoveL Openhole_137, v10, fine, pHeader\WObj:=wobj0;
		MoveL Openhole_138, v10, fine, pHeader\WObj:=wobj0;
		MoveL Openhole_139, v10, fine, pHeader\WObj:=wobj0;
		MoveL Openhole_140, v10, fine, pHeader\WObj:=wobj0;
		MoveL Openhole_141, v10, fine, pHeader\WObj:=wobj0;
		MoveL Openhole_142, v10, fine, pHeader\WObj:=wobj0;
		MoveL Openhole_143, v10, fine, pHeader\WObj:=wobj0;
		MoveL Openhole_144, v10, fine, pHeader\WObj:=wobj0;
		MoveL Openhole_145, v10, fine, pHeader\WObj:=wobj0;
		MoveL Openhole_146, v10, fine, pHeader\WObj:=wobj0;
		MoveL Openhole_147, v10, fine, pHeader\WObj:=wobj0;
		MoveL Openhole_148, v10, fine, pHeader\WObj:=wobj0;
		MoveL Openhole_149, v10, fine, pHeader\WObj:=wobj0;
		MoveL Openhole_150, v10, fine, pHeader\WObj:=wobj0;
		MoveL Openhole_151, v10, fine, pHeader\WObj:=wobj0;
		MoveL Openhole_152, v10, fine, pHeader\WObj:=wobj0;
		MoveL Openhole_153, v10, fine, pHeader\WObj:=wobj0;
		MoveL Openhole_154, v10, fine, pHeader\WObj:=wobj0;
		MoveL Openhole_155, v10, fine, pHeader\WObj:=wobj0;
		MoveL Openhole_156, v10, fine, pHeader\WObj:=wobj0;
		MoveL Openhole_157, v10, fine, pHeader\WObj:=wobj0;
		MoveL Openhole_158, v10, fine, pHeader\WObj:=wobj0;
		MoveL Openhole_159, v10, fine, pHeader\WObj:=wobj0;
		MoveL Openhole_160, v10, fine, pHeader\WObj:=wobj0;
		MoveL Openhole_161, v10, fine, pHeader\WObj:=wobj0;
		MoveL Openhole_162, v10, fine, pHeader\WObj:=wobj0;
		MoveL Openhole_163, v10, fine, pHeader\WObj:=wobj0;
		MoveL Openhole_164, v10, fine, pHeader\WObj:=wobj0;
		MoveL Openhole_165, v10, fine, pHeader\WObj:=wobj0;
		MoveL Openhole_166, v10, fine, pHeader\WObj:=wobj0;
		MoveL Openhole_167, v10, fine, pHeader\WObj:=wobj0;
		MoveL Openhole_168, v10, fine, pHeader\WObj:=wobj0;
		MoveL Openhole_169, v10, fine, pHeader\WObj:=wobj0;
		MoveL Openhole_170, v10, fine, pHeader\WObj:=wobj0;
		MoveL Openhole_171, v10, fine, pHeader\WObj:=wobj0;
		MoveL Openhole_172, v10, fine, pHeader\WObj:=wobj0;
		MoveL Openhole_173, v10, fine, pHeader\WObj:=wobj0;
		MoveL Openhole_174, v10, fine, pHeader\WObj:=wobj0;
		MoveL Openhole_175, v10, fine, pHeader\WObj:=wobj0;
		MoveL Openhole_176, v10, fine, pHeader\WObj:=wobj0;
		MoveL Openhole_177, v10, fine, pHeader\WObj:=wobj0;
		MoveL Openhole_178, v10, fine, pHeader\WObj:=wobj0;
		MoveL Openhole_179, v10, fine, pHeader\WObj:=wobj0;
		MoveL Openhole_180, v10, fine, pHeader\WObj:=wobj0;
		MoveL Openhole_181, v10, fine, pHeader\WObj:=wobj0;
		MoveL Openhole_182, v10, fine, pHeader\WObj:=wobj0;
		MoveL Openhole_183, v10, fine, pHeader\WObj:=wobj0;
		MoveL Openhole_184, v10, fine, pHeader\WObj:=wobj0;
		MoveL Openhole_185, v10, fine, pHeader\WObj:=wobj0;
		MoveL Openhole_186, v10, fine, pHeader\WObj:=wobj0;
		MoveL Openhole_187, v10, fine, pHeader\WObj:=wobj0;
		MoveL Openhole_188, v10, fine, pHeader\WObj:=wobj0;
		MoveL Openhole_189, v10, fine, pHeader\WObj:=wobj0;
		MoveL Openhole_190, v10, fine, pHeader\WObj:=wobj0;
		MoveL Openhole_191, v10, fine, pHeader\WObj:=wobj0;
		MoveL Openhole_192, v10, fine, pHeader\WObj:=wobj0;
		MoveL Openhole_193, v10, fine, pHeader\WObj:=wobj0;
		MoveL Openhole_194, v10, fine, pHeader\WObj:=wobj0;
		MoveL Openhole_195, v10, fine, pHeader\WObj:=wobj0;
		MoveL Openhole_196, v10, fine, pHeader\WObj:=wobj0;
		MoveL Openhole_197, v10, fine, pHeader\WObj:=wobj0;
		MoveL Openhole_198, v10, fine, pHeader\WObj:=wobj0;
		MoveL Openhole_199, v10, fine, pHeader\WObj:=wobj0;
		MoveL Openhole_200, v10, fine, pHeader\WObj:=wobj0;
		MoveL Openhole_201, v10, fine, pHeader\WObj:=wobj0;
		MoveL Openhole_202, v10, fine, pHeader\WObj:=wobj0;
		MoveL Openhole_203, v10, fine, pHeader\WObj:=wobj0;
		MoveL Openhole_204, v10, fine, pHeader\WObj:=wobj0;
		MoveL Openhole_205, v10, fine, pHeader\WObj:=wobj0;
		MoveL Openhole_206, v10, fine, pHeader\WObj:=wobj0;
		MoveL Openhole_207, v10, fine, pHeader\WObj:=wobj0;
		MoveL Openhole_208, v10, fine, pHeader\WObj:=wobj0;
		MoveL Openhole_209, v10, fine, pHeader\WObj:=wobj0;
		MoveL Openhole_210, v10, fine, pHeader\WObj:=wobj0;
		MoveL Openhole_211, v10, fine, pHeader\WObj:=wobj0;
		MoveL Openhole_212, v10, fine, pHeader\WObj:=wobj0;
		MoveL Openhole_213, v10, fine, pHeader\WObj:=wobj0;
		MoveL Openhole_214, v10, fine, pHeader\WObj:=wobj0;
		MoveL Openhole_215, v10, fine, pHeader\WObj:=wobj0;
		MoveL Openhole_216, v10, fine, pHeader\WObj:=wobj0;
		MoveL Openhole_217, v10, fine, pHeader\WObj:=wobj0;
		MoveL Openhole_218, v10, fine, pHeader\WObj:=wobj0;
		MoveL Openhole_219, v10, fine, pHeader\WObj:=wobj0;
		MoveL Openhole_220, v10, fine, pHeader\WObj:=wobj0;
		MoveL Openhole_221, v10, fine, pHeader\WObj:=wobj0;
		MoveL Openhole_222, v10, fine, pHeader\WObj:=wobj0;
		MoveL Openhole_223, v10, fine, pHeader\WObj:=wobj0;
		MoveL Openhole_224, v10, fine, pHeader\WObj:=wobj0;
		MoveL Openhole_225, v10, fine, pHeader\WObj:=wobj0;
		MoveL Openhole_226, v10, fine, pHeader\WObj:=wobj0;
		MoveL Openhole_227, v10, fine, pHeader\WObj:=wobj0;
		MoveL Openhole_228, v10, fine, pHeader\WObj:=wobj0;
		MoveL Openhole_229, v10, fine, pHeader\WObj:=wobj0;
		MoveL Openhole_230, v10, fine, pHeader\WObj:=wobj0;
		MoveL Openhole_231, v10, fine, pHeader\WObj:=wobj0;
		MoveL Openhole_232, v10, fine, pHeader\WObj:=wobj0;
		MoveL Openhole_233, v10, fine, pHeader\WObj:=wobj0;
		MoveL Openhole_234, v10, fine, pHeader\WObj:=wobj0;
		MoveL Openhole_235, v10, fine, pHeader\WObj:=wobj0;
		MoveL Openhole_236, v10, fine, pHeader\WObj:=wobj0;
		MoveL Openhole_237, v10, fine, pHeader\WObj:=wobj0;
		MoveL Openhole_238, v10, fine, pHeader\WObj:=wobj0;
		MoveL Openhole_239, v10, fine, pHeader\WObj:=wobj0;
		MoveL Openhole_240, v10, fine, pHeader\WObj:=wobj0;
		MoveL Openhole_241, v10, fine, pHeader\WObj:=wobj0;
		MoveL Openhole_242, v10, fine, pHeader\WObj:=wobj0;
		MoveL Openhole_243, v10, fine, pHeader\WObj:=wobj0;
		MoveL Openhole_244, v10, fine, pHeader\WObj:=wobj0;
		MoveL Openhole_245, v10, fine, pHeader\WObj:=wobj0;
		MoveL Openhole_246, v10, fine, pHeader\WObj:=wobj0;
		MoveL Openhole_247, v10, fine, pHeader\WObj:=wobj0;
		MoveL Openhole_248, v10, fine, pHeader\WObj:=wobj0;
		MoveL Openhole_249, v10, fine, pHeader\WObj:=wobj0;
		MoveL Openhole_250, v10, fine, pHeader\WObj:=wobj0;
		MoveL Openhole_251, v10, fine, pHeader\WObj:=wobj0;
		MoveL Openhole_252, v10, fine, pHeader\WObj:=wobj0;
		MoveL Openhole_253, v10, fine, pHeader\WObj:=wobj0;
		MoveL Openhole_254, v10, fine, pHeader\WObj:=wobj0;
		MoveL Openhole_255, v10, fine, pHeader\WObj:=wobj0;
		MoveL Openhole_256, v10, fine, pHeader\WObj:=wobj0;
		MoveL Openhole_257, v10, fine, pHeader\WObj:=wobj0;
		MoveL Openhole_258, v10, fine, pHeader\WObj:=wobj0;
		MoveL Openhole_259, v10, fine, pHeader\WObj:=wobj0;
		MoveL Openhole_260, v10, fine, pHeader\WObj:=wobj0;
		MoveL Openhole_261, v10, fine, pHeader\WObj:=wobj0;
		MoveL Openhole_262, v10, fine, pHeader\WObj:=wobj0;
		MoveL Openhole_263, v10, fine, pHeader\WObj:=wobj0;
		MoveL Openhole_264, v10, fine, pHeader\WObj:=wobj0;
		MoveL Openhole_265, v10, fine, pHeader\WObj:=wobj0;
		MoveL Openhole_266, v10, fine, pHeader\WObj:=wobj0;
		MoveL Openhole_267, v10, fine, pHeader\WObj:=wobj0;
		MoveL Openhole_268, v10, fine, pHeader\WObj:=wobj0;
		MoveL Openhole_269, v10, fine, pHeader\WObj:=wobj0;
		MoveL Openhole_270, v10, fine, pHeader\WObj:=wobj0;
		MoveL Openhole_271, v10, fine, pHeader\WObj:=wobj0;
		MoveL Openhole_272, v10, fine, pHeader\WObj:=wobj0;
		MoveL Openhole_273, v10, fine, pHeader\WObj:=wobj0;
		MoveL Openhole_274, v10, fine, pHeader\WObj:=wobj0;
		MoveL Openhole_275, v10, fine, pHeader\WObj:=wobj0;
		MoveL Openhole_276, v10, fine, pHeader\WObj:=wobj0;
		MoveL Openhole_277, v10, fine, pHeader\WObj:=wobj0;
		MoveL Openhole_278, v10, fine, pHeader\WObj:=wobj0;
		MoveL Openhole_279, v10, fine, pHeader\WObj:=wobj0;
		MoveL Openhole_280, v10, fine, pHeader\WObj:=wobj0;
		MoveL Openhole_281, v10, fine, pHeader\WObj:=wobj0;
		MoveL Openhole_282, v10, fine, pHeader\WObj:=wobj0;
		MoveL Openhole_283, v10, fine, pHeader\WObj:=wobj0;
		MoveL Openhole_284, v10, fine, pHeader\WObj:=wobj0;
		MoveL Openhole_285, v10, fine, pHeader\WObj:=wobj0;
		MoveL Openhole_286, v10, fine, pHeader\WObj:=wobj0;
		MoveL Openhole_287, v10, fine, pHeader\WObj:=wobj0;
		MoveL Openhole_288, v10, fine, pHeader\WObj:=wobj0;
		MoveL Openhole_289, v10, fine, pHeader\WObj:=wobj0;
		MoveL Openhole_290, v10, fine, pHeader\WObj:=wobj0;
		MoveL Openhole_291, v10, fine, pHeader\WObj:=wobj0;
		MoveL Openhole_292, v10, fine, pHeader\WObj:=wobj0;
		MoveL Openhole_293, v10, fine, pHeader\WObj:=wobj0;
		MoveL Openhole_294, v10, fine, pHeader\WObj:=wobj0;
		MoveL Openhole_295, v10, fine, pHeader\WObj:=wobj0;
		MoveL Openhole_296, v10, fine, pHeader\WObj:=wobj0;
		MoveL Openhole_297, v10, fine, pHeader\WObj:=wobj0;
		MoveL Openhole_298, v10, fine, pHeader\WObj:=wobj0;
		MoveL Openhole_299, v10, fine, pHeader\WObj:=wobj0;
		MoveL Openhole_300, v10, fine, pHeader\WObj:=wobj0;
		MoveL Openhole_301, v10, fine, pHeader\WObj:=wobj0;
		MoveL Openhole_302, v10, fine, pHeader\WObj:=wobj0;
		MoveL Openhole_303, v10, fine, pHeader\WObj:=wobj0;
		MoveL Openhole_304, v10, fine, pHeader\WObj:=wobj0;
		MoveL Openhole_305, v10, fine, pHeader\WObj:=wobj0;
		MoveL Openhole_306, v10, fine, pHeader\WObj:=wobj0;
		MoveL Openhole_307, v10, fine, pHeader\WObj:=wobj0;
		MoveL Openhole_308, v10, fine, pHeader\WObj:=wobj0;
		MoveL Openhole_309, v10, fine, pHeader\WObj:=wobj0;
		MoveL Openhole_310, v10, fine, pHeader\WObj:=wobj0;
		MoveL Openhole_311, v10, fine, pHeader\WObj:=wobj0;
		MoveL Openhole_312, v10, fine, pHeader\WObj:=wobj0;
		MoveL Openhole_313, v10, fine, pHeader\WObj:=wobj0;
		MoveL Openhole_314, v10, fine, pHeader\WObj:=wobj0;
		MoveL Openhole_315, v10, fine, pHeader\WObj:=wobj0;
		MoveL Openhole_316, v10, fine, pHeader\WObj:=wobj0;
		MoveL Openhole_317, v10, fine, pHeader\WObj:=wobj0;
		MoveL Openhole_318, v10, fine, pHeader\WObj:=wobj0;
		MoveL Openhole_319, v10, fine, pHeader\WObj:=wobj0;
		MoveL Openhole_320, v10, fine, pHeader\WObj:=wobj0;
		MoveL Openhole_321, v10, fine, pHeader\WObj:=wobj0;
		MoveL Openhole_322, v10, fine, pHeader\WObj:=wobj0;
		MoveL Openhole_323, v10, fine, pHeader\WObj:=wobj0;
		MoveL Openhole_324, v10, fine, pHeader\WObj:=wobj0;
		MoveL Openhole_325, v10, fine, pHeader\WObj:=wobj0;
		MoveL Openhole_326, v10, fine, pHeader\WObj:=wobj0;
		MoveL Openhole_327, v10, fine, pHeader\WObj:=wobj0;
		MoveL Openhole_328, v10, fine, pHeader\WObj:=wobj0;
		MoveL Openhole_329, v10, fine, pHeader\WObj:=wobj0;
		MoveL Openhole_330, v10, fine, pHeader\WObj:=wobj0;
		MoveL Openhole_331, v10, fine, pHeader\WObj:=wobj0;
		MoveL Openhole_332, v10, fine, pHeader\WObj:=wobj0;
		MoveL Openhole_333, v10, fine, pHeader\WObj:=wobj0;
		MoveL Openhole_334, v10, fine, pHeader\WObj:=wobj0;
		MoveL Openhole_335, v10, fine, pHeader\WObj:=wobj0;
		MoveL Openhole_336, v10, fine, pHeader\WObj:=wobj0;
		MoveL Openhole_337, v10, fine, pHeader\WObj:=wobj0;
		MoveL Openhole_338, v10, fine, pHeader\WObj:=wobj0;
		MoveL Openhole_339, v10, fine, pHeader\WObj:=wobj0;
		MoveL Openhole_340, v10, fine, pHeader\WObj:=wobj0;
		MoveL Openhole_341, v10, fine, pHeader\WObj:=wobj0;
		MoveL Openhole_342, v10, fine, pHeader\WObj:=wobj0;
		MoveL Openhole_343, v10, fine, pHeader\WObj:=wobj0;
		MoveL Openhole_344, v10, fine, pHeader\WObj:=wobj0;
		MoveL Openhole_345, v10, fine, pHeader\WObj:=wobj0;
		MoveL Openhole_346, v10, fine, pHeader\WObj:=wobj0;
		MoveL Openhole_347, v10, fine, pHeader\WObj:=wobj0;
		MoveL Openhole_348, v10, fine, pHeader\WObj:=wobj0;
		MoveL Openhole_349, v10, fine, pHeader\WObj:=wobj0;
		MoveL Openhole_350, v10, fine, pHeader\WObj:=wobj0;
		MoveL Openhole_351, v10, fine, pHeader\WObj:=wobj0;
		MoveL Openhole_352, v10, fine, pHeader\WObj:=wobj0;
		MoveL Openhole_353, v10, fine, pHeader\WObj:=wobj0;
		MoveL Openhole_354, v10, fine, pHeader\WObj:=wobj0;
		MoveL Openhole_355, v10, fine, pHeader\WObj:=wobj0;
		MoveL Openhole_356, v10, fine, pHeader\WObj:=wobj0;
		MoveL Openhole_357, v10, fine, pHeader\WObj:=wobj0;
		MoveL Openhole_358, v10, fine, pHeader\WObj:=wobj0;
		MoveL Openhole_359, v10, fine, pHeader\WObj:=wobj0;
		MoveL Openhole_360, v10, fine, pHeader\WObj:=wobj0;
		MoveL Openhole_361, v10, fine, pHeader\WObj:=wobj0;
		MoveL Openhole_362, v10, fine, pHeader\WObj:=wobj0;
		MoveL Openhole_363, v10, fine, pHeader\WObj:=wobj0;
		MoveL Openhole_364, v10, fine, pHeader\WObj:=wobj0;
		MoveL Openhole_365, v10, fine, pHeader\WObj:=wobj0;
		MoveL Openhole_366, v10, fine, pHeader\WObj:=wobj0;
		MoveL Openhole_367, v10, fine, pHeader\WObj:=wobj0;
		MoveL Openhole_368, v10, fine, pHeader\WObj:=wobj0;
		MoveL Openhole_369, v10, fine, pHeader\WObj:=wobj0;
		MoveL Openhole_370, v10, fine, pHeader\WObj:=wobj0;
		MoveL Openhole_371, v10, fine, pHeader\WObj:=wobj0;
		MoveL Openhole_372, v10, fine, pHeader\WObj:=wobj0;
		MoveL Openhole_373, v10, fine, pHeader\WObj:=wobj0;
		MoveL Openhole_374, v10, fine, pHeader\WObj:=wobj0;
		MoveL Openhole_375, v10, fine, pHeader\WObj:=wobj0;
		MoveL Openhole_376, v10, fine, pHeader\WObj:=wobj0;
		MoveL Openhole_377, v10, fine, pHeader\WObj:=wobj0;
		MoveL Openhole_378, v10, fine, pHeader\WObj:=wobj0;
		MoveL Openhole_379, v10, fine, pHeader\WObj:=wobj0;
		MoveL Openhole_380, v10, fine, pHeader\WObj:=wobj0;
		MoveL Openhole_381, v10, fine, pHeader\WObj:=wobj0;
		MoveL Openhole_382, v10, fine, pHeader\WObj:=wobj0;
		MoveL Openhole_383, v10, fine, pHeader\WObj:=wobj0;
		MoveL Openhole_384, v10, fine, pHeader\WObj:=wobj0;
		MoveL Openhole_385, v10, fine, pHeader\WObj:=wobj0;
		MoveL Openhole_386, v10, fine, pHeader\WObj:=wobj0;
		MoveL Openhole_387, v10, fine, pHeader\WObj:=wobj0;
		MoveL Openhole_388, v10, fine, pHeader\WObj:=wobj0;
		MoveL Openhole_389, v10, fine, pHeader\WObj:=wobj0;
		MoveL Openhole_390, v10, fine, pHeader\WObj:=wobj0;
		MoveL Openhole_391, v10, fine, pHeader\WObj:=wobj0;
		MoveL Openhole_392, v10, fine, pHeader\WObj:=wobj0;
		MoveL Openhole_393, v10, fine, pHeader\WObj:=wobj0;
		MoveL Openhole_394, v10, fine, pHeader\WObj:=wobj0;
		MoveL Openhole_395, v10, fine, pHeader\WObj:=wobj0;
		MoveL Openhole_396, v10, fine, pHeader\WObj:=wobj0;
		MoveL Openhole_397, v10, fine, pHeader\WObj:=wobj0;
		MoveL Openhole_398, v10, fine, pHeader\WObj:=wobj0;
		MoveL Openhole_399, v10, fine, pHeader\WObj:=wobj0;
		MoveL Openhole_400, v10, fine, pHeader\WObj:=wobj0;
		MoveL Openhole_401, v10, fine, pHeader\WObj:=wobj0;
		MoveL Openhole_402, v10, fine, pHeader\WObj:=wobj0;
		MoveL Openhole_403, v10, fine, pHeader\WObj:=wobj0;
		MoveL Openhole_404, v10, fine, pHeader\WObj:=wobj0;
		MoveL Openhole_405, v10, fine, pHeader\WObj:=wobj0;
		MoveL Openhole_406, v10, fine, pHeader\WObj:=wobj0;
		MoveL Openhole_407, v10, fine, pHeader\WObj:=wobj0;
		MoveL Openhole_408, v10, fine, pHeader\WObj:=wobj0;
		MoveL Openhole_409, v10, fine, pHeader\WObj:=wobj0;
		MoveL Openhole_410, v10, fine, pHeader\WObj:=wobj0;
		MoveL Openhole_411, v10, fine, pHeader\WObj:=wobj0;
		MoveL Openhole_412, v10, fine, pHeader\WObj:=wobj0;
		MoveL Openhole_413, v10, fine, pHeader\WObj:=wobj0;
		MoveL Openhole_414, v10, fine, pHeader\WObj:=wobj0;
		MoveL Openhole_415, v10, fine, pHeader\WObj:=wobj0;
		MoveL Openhole_416, v10, fine, pHeader\WObj:=wobj0;
		MoveL Openhole_417, v10, fine, pHeader\WObj:=wobj0;
		MoveL Openhole_418, v10, fine, pHeader\WObj:=wobj0;
		MoveL Openhole_419, v10, fine, pHeader\WObj:=wobj0;
		MoveL Openhole_420, v10, fine, pHeader\WObj:=wobj0;
		MoveL Openhole_421, v10, fine, pHeader\WObj:=wobj0;
		MoveL Openhole_422, v10, fine, pHeader\WObj:=wobj0;
		MoveL Openhole_423, v10, fine, pHeader\WObj:=wobj0;
		MoveL Openhole_424, v10, fine, pHeader\WObj:=wobj0;
		MoveL Openhole_425, v10, fine, pHeader\WObj:=wobj0;
		MoveL Openhole_426, v10, fine, pHeader\WObj:=wobj0;
		MoveL Openhole_427, v10, fine, pHeader\WObj:=wobj0;
		MoveL Openhole_428, v10, fine, pHeader\WObj:=wobj0;
		MoveL Openhole_429, v10, fine, pHeader\WObj:=wobj0;
		MoveL Openhole_430, v10, fine, pHeader\WObj:=wobj0;
		MoveL Openhole_431, v10, fine, pHeader\WObj:=wobj0;
		MoveL Openhole_432, v10, fine, pHeader\WObj:=wobj0;
		MoveL Openhole_433, v10, fine, pHeader\WObj:=wobj0;
		MoveL Openhole_434, v10, fine, pHeader\WObj:=wobj0;
		MoveL Openhole_435, v10, fine, pHeader\WObj:=wobj0;
		MoveL Openhole_436, v10, fine, pHeader\WObj:=wobj0;
		MoveL Openhole_437, v10, fine, pHeader\WObj:=wobj0;
		MoveL Openhole_438, v10, fine, pHeader\WObj:=wobj0;
		MoveL Openhole_439, v10, fine, pHeader\WObj:=wobj0;
		MoveL Openhole_440, v10, fine, pHeader\WObj:=wobj0;
		MoveL Openhole_441, v10, fine, pHeader\WObj:=wobj0;
		MoveL Openhole_442, v10, fine, pHeader\WObj:=wobj0;
		MoveL Openhole_443, v10, fine, pHeader\WObj:=wobj0;
		MoveL Openhole_444, v10, fine, pHeader\WObj:=wobj0;
		MoveL Openhole_445, v10, fine, pHeader\WObj:=wobj0;
		MoveL Openhole_446, v10, fine, pHeader\WObj:=wobj0;
		MoveL Openhole_447, v10, fine, pHeader\WObj:=wobj0;
		MoveL Openhole_448, v10, fine, pHeader\WObj:=wobj0;
		MoveL Openhole_449, v10, fine, pHeader\WObj:=wobj0;
		MoveL Openhole_450, v10, fine, pHeader\WObj:=wobj0;
		MoveL Openhole_451, v10, fine, pHeader\WObj:=wobj0;
		MoveL Openhole_452, v10, fine, pHeader\WObj:=wobj0;
		MoveL Openhole_453, v10, fine, pHeader\WObj:=wobj0;
		MoveL Openhole_454, v10, fine, pHeader\WObj:=wobj0;
		MoveL Openhole_455, v10, fine, pHeader\WObj:=wobj0;
		MoveL Openhole_456, v10, fine, pHeader\WObj:=wobj0;
		MoveL Openhole_457, v10, fine, pHeader\WObj:=wobj0;
		MoveL Openhole_458, v10, fine, pHeader\WObj:=wobj0;
		MoveL Openhole_459, v10, fine, pHeader\WObj:=wobj0;
		MoveL Openhole_460, v10, fine, pHeader\WObj:=wobj0;
		MoveL Openhole_461, v10, fine, pHeader\WObj:=wobj0;
		MoveL Openhole_462, v10, fine, pHeader\WObj:=wobj0;
		MoveL Openhole_463, v10, fine, pHeader\WObj:=wobj0;
		MoveL Openhole_464, v10, fine, pHeader\WObj:=wobj0;
		MoveL Openhole_465, v10, fine, pHeader\WObj:=wobj0;
		MoveL Openhole_466, v10, fine, pHeader\WObj:=wobj0;
		MoveL Openhole_467, v10, fine, pHeader\WObj:=wobj0;
		MoveL Openhole_468, v10, fine, pHeader\WObj:=wobj0;
		MoveL Openhole_469, v10, fine, pHeader\WObj:=wobj0;
		MoveL Openhole_470, v10, fine, pHeader\WObj:=wobj0;
		MoveL Openhole_471, v10, fine, pHeader\WObj:=wobj0;
		MoveL Openhole_472, v10, fine, pHeader\WObj:=wobj0;
		MoveL Openhole_473, v10, fine, pHeader\WObj:=wobj0;
		MoveL Openhole_474, v10, fine, pHeader\WObj:=wobj0;
		MoveL Openhole_475, v10, fine, pHeader\WObj:=wobj0;
		MoveL Openhole_476, v10, fine, pHeader\WObj:=wobj0;
		MoveL Openhole_477, v10, fine, pHeader\WObj:=wobj0;
		MoveL Openhole_478, v10, fine, pHeader\WObj:=wobj0;
		MoveL Openhole_479, v10, fine, pHeader\WObj:=wobj0;
		MoveL Openhole_480, v10, fine, pHeader\WObj:=wobj0;
		MoveL Openhole_481, v10, fine, pHeader\WObj:=wobj0;
		MoveL Openhole_482, v10, fine, pHeader\WObj:=wobj0;
		MoveL Openhole_483, v10, fine, pHeader\WObj:=wobj0;
		MoveL Openhole_484, v10, fine, pHeader\WObj:=wobj0;
		MoveL Openhole_485, v10, fine, pHeader\WObj:=wobj0;
		MoveL Openhole_486, v10, fine, pHeader\WObj:=wobj0;
		MoveL Openhole_487, v10, fine, pHeader\WObj:=wobj0;
		MoveL Openhole_488, v10, fine, pHeader\WObj:=wobj0;
		MoveL Openhole_489, v10, fine, pHeader\WObj:=wobj0;
		MoveL Openhole_490, v10, fine, pHeader\WObj:=wobj0;
		MoveL Openhole_491, v10, fine, pHeader\WObj:=wobj0;
		MoveL Openhole_492, v10, fine, pHeader\WObj:=wobj0;
		MoveL Openhole_493, v10, fine, pHeader\WObj:=wobj0;
		MoveL Openhole_494, v10, fine, pHeader\WObj:=wobj0;
		MoveL Openhole_495, v10, fine, pHeader\WObj:=wobj0;
		MoveL Openhole_496, v10, fine, pHeader\WObj:=wobj0;
		MoveL Openhole_497, v10, fine, pHeader\WObj:=wobj0;
		MoveL Openhole_498, v10, fine, pHeader\WObj:=wobj0;
		MoveL Openhole_499, v10, fine, pHeader\WObj:=wobj0;
		MoveL Openhole_500, v10, fine, pHeader\WObj:=wobj0;
		MoveL Openhole_501, v10, fine, pHeader\WObj:=wobj0;
		MoveL Openhole_502, v10, fine, pHeader\WObj:=wobj0;
		MoveL Openhole_503, v10, fine, pHeader\WObj:=wobj0;
		MoveL Openhole_504, v10, fine, pHeader\WObj:=wobj0;
		MoveL Openhole_505, v10, fine, pHeader\WObj:=wobj0;
		MoveL Openhole_506, v10, fine, pHeader\WObj:=wobj0;
		MoveL Openhole_507, v10, fine, pHeader\WObj:=wobj0;
		MoveL Openhole_508, v10, fine, pHeader\WObj:=wobj0;
		MoveL Openhole_509, v10, fine, pHeader\WObj:=wobj0;
		MoveL Openhole_510, v10, fine, pHeader\WObj:=wobj0;
		MoveL Openhole_511, v10, fine, pHeader\WObj:=wobj0;
		MoveL Openhole_512, v10, fine, pHeader\WObj:=wobj0;
		MoveL Openhole_513, v10, fine, pHeader\WObj:=wobj0;
		MoveL Openhole_514, v10, fine, pHeader\WObj:=wobj0;
		MoveL Openhole_515, v10, fine, pHeader\WObj:=wobj0;
		MoveL Openhole_516, v10, fine, pHeader\WObj:=wobj0;
		MoveL Openhole_517, v10, fine, pHeader\WObj:=wobj0;
		MoveL Openhole_518, v10, fine, pHeader\WObj:=wobj0;
		MoveL Openhole_519, v10, fine, pHeader\WObj:=wobj0;
		MoveL Openhole_520, v10, fine, pHeader\WObj:=wobj0;
		MoveL Openhole_521, v10, fine, pHeader\WObj:=wobj0;
		MoveL Openhole_522, v10, fine, pHeader\WObj:=wobj0;
		MoveL Openhole_523, v10, fine, pHeader\WObj:=wobj0;
		MoveL Openhole_524, v10, fine, pHeader\WObj:=wobj0;
		MoveL Openhole_525, v10, fine, pHeader\WObj:=wobj0;
		MoveL Openhole_526, v10, fine, pHeader\WObj:=wobj0;
		MoveL Openhole_527, v10, fine, pHeader\WObj:=wobj0;
		MoveL Openhole_528, v10, fine, pHeader\WObj:=wobj0;
		MoveL Openhole_529, v10, fine, pHeader\WObj:=wobj0;
		MoveL Openhole_530, v10, fine, pHeader\WObj:=wobj0;
		MoveL Openhole_531, v10, fine, pHeader\WObj:=wobj0;
		MoveL Openhole_532, v10, fine, pHeader\WObj:=wobj0;
		MoveL Openhole_533, v10, fine, pHeader\WObj:=wobj0;
		MoveL Openhole_534, v10, fine, pHeader\WObj:=wobj0;
		MoveL Openhole_535, v10, fine, pHeader\WObj:=wobj0;
		MoveL Openhole_536, v10, fine, pHeader\WObj:=wobj0;
		MoveL Openhole_537, v10, fine, pHeader\WObj:=wobj0;
		MoveL Openhole_538, v10, fine, pHeader\WObj:=wobj0;
		MoveL Openhole_539, v10, fine, pHeader\WObj:=wobj0;
		MoveL Openhole_540, v10, fine, pHeader\WObj:=wobj0;
		MoveL Openhole_541, v10, fine, pHeader\WObj:=wobj0;
		MoveL Openhole_542, v10, fine, pHeader\WObj:=wobj0;
		MoveL Openhole_543, v10, fine, pHeader\WObj:=wobj0;
		MoveL Openhole_544, v10, fine, pHeader\WObj:=wobj0;
		MoveL Openhole_545, v10, fine, pHeader\WObj:=wobj0;
		MoveL Openhole_546, v10, fine, pHeader\WObj:=wobj0;
		MoveL Openhole_547, v10, fine, pHeader\WObj:=wobj0;
		MoveL Openhole_548, v10, fine, pHeader\WObj:=wobj0;
		MoveL Openhole_549, v10, fine, pHeader\WObj:=wobj0;
		MoveL Openhole_550, v10, fine, pHeader\WObj:=wobj0;
		MoveL Openhole_551, v10, fine, pHeader\WObj:=wobj0;
		MoveL Openhole_552, v10, fine, pHeader\WObj:=wobj0;
		MoveL Openhole_553, v10, fine, pHeader\WObj:=wobj0;
		MoveL Openhole_554, v10, fine, pHeader\WObj:=wobj0;
		MoveL Openhole_555, v10, fine, pHeader\WObj:=wobj0;
		MoveL Openhole_556, v10, fine, pHeader\WObj:=wobj0;
		MoveL Openhole_557, v10, fine, pHeader\WObj:=wobj0;
		MoveL Openhole_558, v10, fine, pHeader\WObj:=wobj0;
		MoveL Openhole_559, v10, fine, pHeader\WObj:=wobj0;
		MoveL Openhole_560, v10, fine, pHeader\WObj:=wobj0;
		MoveL Openhole_561, v10, fine, pHeader\WObj:=wobj0;
		MoveL Openhole_562, v10, fine, pHeader\WObj:=wobj0;
		MoveL Openhole_563, v10, fine, pHeader\WObj:=wobj0;
		MoveL Openhole_564, v10, fine, pHeader\WObj:=wobj0;
		MoveL Openhole_565, v10, fine, pHeader\WObj:=wobj0;
		MoveL Openhole_566, v10, fine, pHeader\WObj:=wobj0;
		MoveL Openhole_567, v10, fine, pHeader\WObj:=wobj0;
		MoveL Openhole_568, v10, fine, pHeader\WObj:=wobj0;
		MoveL Openhole_569, v10, fine, pHeader\WObj:=wobj0;
		MoveL Openhole_570, v10, fine, pHeader\WObj:=wobj0;
		MoveL Openhole_571, v10, fine, pHeader\WObj:=wobj0;
		MoveL Openhole_572, v10, fine, pHeader\WObj:=wobj0;
		MoveL Openhole_573, v10, fine, pHeader\WObj:=wobj0;
		MoveL Openhole_574, v10, fine, pHeader\WObj:=wobj0;
		MoveL Openhole_575, v10, fine, pHeader\WObj:=wobj0;
		MoveL Openhole_576, v10, fine, pHeader\WObj:=wobj0;
		MoveL Openhole_577, v10, fine, pHeader\WObj:=wobj0;
		MoveL Openhole_578, v10, fine, pHeader\WObj:=wobj0;
		MoveL Openhole_579, v10, fine, pHeader\WObj:=wobj0;
		MoveL Openhole_580, v10, fine, pHeader\WObj:=wobj0;
		MoveL Openhole_581, v10, fine, pHeader\WObj:=wobj0;
		MoveL Openhole_582, v10, fine, pHeader\WObj:=wobj0;
		MoveL Openhole_583, v10, fine, pHeader\WObj:=wobj0;
		MoveL Openhole_584, v10, fine, pHeader\WObj:=wobj0;
		MoveL Openhole_585, v10, fine, pHeader\WObj:=wobj0;
		MoveL Openhole_586, v10, fine, pHeader\WObj:=wobj0;
		MoveL Openhole_587, v10, fine, pHeader\WObj:=wobj0;
		MoveL Openhole_588, v10, fine, pHeader\WObj:=wobj0;
		MoveL Openhole_589, v10, fine, pHeader\WObj:=wobj0;
		MoveL Openhole_590, v10, fine, pHeader\WObj:=wobj0;
		MoveL Openhole_591, v10, fine, pHeader\WObj:=wobj0;
		MoveL Openhole_592, v10, fine, pHeader\WObj:=wobj0;
		MoveL Openhole_593, v10, fine, pHeader\WObj:=wobj0;
		MoveL Openhole_594, v10, fine, pHeader\WObj:=wobj0;
		MoveL Openhole_595, v10, fine, pHeader\WObj:=wobj0;
		MoveL Openhole_596, v10, fine, pHeader\WObj:=wobj0;
		MoveL Openhole_597, v10, fine, pHeader\WObj:=wobj0;
		MoveL Openhole_598, v10, fine, pHeader\WObj:=wobj0;
		MoveL Openhole_599, v10, fine, pHeader\WObj:=wobj0;
		MoveL Openhole_600, v10, fine, pHeader\WObj:=wobj0;
		MoveL Openhole_601, v10, fine, pHeader\WObj:=wobj0;
		MoveL Openhole_602, v10, fine, pHeader\WObj:=wobj0;
		MoveL Openhole_603, v10, fine, pHeader\WObj:=wobj0;
		MoveL Openhole_604, v10, fine, pHeader\WObj:=wobj0;
		MoveL Openhole_605, v10, fine, pHeader\WObj:=wobj0;
		MoveL Openhole_606, v10, fine, pHeader\WObj:=wobj0;
		MoveL Openhole_607, v10, fine, pHeader\WObj:=wobj0;
		MoveL Openhole_608, v10, fine, pHeader\WObj:=wobj0;
		MoveL Openhole_609, v10, fine, pHeader\WObj:=wobj0;
		MoveL Openhole_610, v10, fine, pHeader\WObj:=wobj0;
		MoveL Openhole_611, v10, fine, pHeader\WObj:=wobj0;
		MoveL Openhole_612, v10, fine, pHeader\WObj:=wobj0;
		MoveL Openhole_613, v10, fine, pHeader\WObj:=wobj0;
		MoveL Openhole_614, v10, fine, pHeader\WObj:=wobj0;
		MoveL Openhole_615, v10, fine, pHeader\WObj:=wobj0;
		MoveL Openhole_616, v10, fine, pHeader\WObj:=wobj0;
		MoveL Openhole_617, v10, fine, pHeader\WObj:=wobj0;
		MoveL Openhole_618, v10, fine, pHeader\WObj:=wobj0;
		MoveL Openhole_619, v10, fine, pHeader\WObj:=wobj0;
		MoveL Openhole_620, v10, fine, pHeader\WObj:=wobj0;
		MoveL Openhole_621, v10, fine, pHeader\WObj:=wobj0;
		MoveL Openhole_622, v10, fine, pHeader\WObj:=wobj0;
		MoveL Openhole_623, v10, fine, pHeader\WObj:=wobj0;
		MoveL Openhole_624, v10, fine, pHeader\WObj:=wobj0;
		MoveL Openhole_625, v10, fine, pHeader\WObj:=wobj0;
		MoveL Openhole_626, v10, fine, pHeader\WObj:=wobj0;
		MoveL Openhole_627, v10, fine, pHeader\WObj:=wobj0;
		MoveL Openhole_628, v10, fine, pHeader\WObj:=wobj0;
		MoveL Openhole_629, v10, fine, pHeader\WObj:=wobj0;
		MoveL Openhole_630, v10, fine, pHeader\WObj:=wobj0;
		MoveL Openhole_631, v10, fine, pHeader\WObj:=wobj0;
		MoveL Openhole_632, v10, fine, pHeader\WObj:=wobj0;
		MoveL Openhole_633, v10, fine, pHeader\WObj:=wobj0;
		MoveL Openhole_634, v10, fine, pHeader\WObj:=wobj0;
		MoveL Openhole_635, v10, fine, pHeader\WObj:=wobj0;
		MoveL Openhole_636, v10, fine, pHeader\WObj:=wobj0;
		MoveL Openhole_637, v10, fine, pHeader\WObj:=wobj0;
		MoveL Openhole_638, v10, fine, pHeader\WObj:=wobj0;
		MoveL Openhole_639, v10, fine, pHeader\WObj:=wobj0;
		MoveL Openhole_640, v10, fine, pHeader\WObj:=wobj0;
		MoveL Openhole_641, v10, fine, pHeader\WObj:=wobj0;
		MoveL Openhole_642, v10, fine, pHeader\WObj:=wobj0;
		MoveL Openhole_643, v10, fine, pHeader\WObj:=wobj0;
		MoveL Openhole_644, v10, fine, pHeader\WObj:=wobj0;
		MoveL Openhole_645, v10, fine, pHeader\WObj:=wobj0;
		MoveL Openhole_646, v10, fine, pHeader\WObj:=wobj0;
		MoveL Openhole_647, v10, fine, pHeader\WObj:=wobj0;
		MoveL Openhole_648, v10, fine, pHeader\WObj:=wobj0;
		MoveL Openhole_649, v10, fine, pHeader\WObj:=wobj0;
		MoveL Openhole_650, v10, fine, pHeader\WObj:=wobj0;
		MoveL Openhole_651, v10, fine, pHeader\WObj:=wobj0;
		MoveL Openhole_652, v10, fine, pHeader\WObj:=wobj0;
		MoveL Openhole_653, v10, fine, pHeader\WObj:=wobj0;
		MoveL Openhole_654, v10, fine, pHeader\WObj:=wobj0;
		MoveL Openhole_655, v10, fine, pHeader\WObj:=wobj0;
		MoveL Openhole_656, v10, fine, pHeader\WObj:=wobj0;
		MoveL Openhole_657, v10, fine, pHeader\WObj:=wobj0;
		MoveL Openhole_658, v10, fine, pHeader\WObj:=wobj0;
		MoveL Openhole_659, v10, fine, pHeader\WObj:=wobj0;
		MoveL Openhole_660, v10, fine, pHeader\WObj:=wobj0;
		MoveL Openhole_661, v10, fine, pHeader\WObj:=wobj0;
		MoveL Openhole_662, v10, fine, pHeader\WObj:=wobj0;
		MoveL Openhole_663, v10, fine, pHeader\WObj:=wobj0;
		MoveL Openhole_664, v10, fine, pHeader\WObj:=wobj0;
		MoveL Openhole_665, v10, fine, pHeader\WObj:=wobj0;
		MoveL Openhole_666, v10, fine, pHeader\WObj:=wobj0;
		MoveL Openhole_667, v10, fine, pHeader\WObj:=wobj0;
		MoveL Openhole_668, v10, fine, pHeader\WObj:=wobj0;
		MoveL Openhole_669, v10, fine, pHeader\WObj:=wobj0;
		MoveL Openhole_670, v10, fine, pHeader\WObj:=wobj0;
		MoveL Openhole_671, v10, fine, pHeader\WObj:=wobj0;
		MoveL Openhole_672, v10, fine, pHeader\WObj:=wobj0;
		MoveL Openhole_673, v10, fine, pHeader\WObj:=wobj0;
		MoveL Openhole_674, v10, fine, pHeader\WObj:=wobj0;
		MoveL Openhole_675, v10, fine, pHeader\WObj:=wobj0;
		MoveL Openhole_676, v10, fine, pHeader\WObj:=wobj0;
		MoveL Openhole_677, v10, fine, pHeader\WObj:=wobj0;
		MoveL Openhole_678, v10, fine, pHeader\WObj:=wobj0;
		MoveL Openhole_679, v10, fine, pHeader\WObj:=wobj0;
		MoveL Openhole_680, v10, fine, pHeader\WObj:=wobj0;
		MoveL Openhole_681, v10, fine, pHeader\WObj:=wobj0;
		MoveL Openhole_682, v10, fine, pHeader\WObj:=wobj0;
		MoveL Openhole_683, v10, fine, pHeader\WObj:=wobj0;
		MoveL Openhole_684, v10, fine, pHeader\WObj:=wobj0;
		MoveL Openhole_685, v10, fine, pHeader\WObj:=wobj0;
		MoveL Openhole_686, v10, fine, pHeader\WObj:=wobj0;
		MoveL Openhole_687, v10, fine, pHeader\WObj:=wobj0;
		MoveL Openhole_688, v10, fine, pHeader\WObj:=wobj0;
		MoveL Openhole_689, v10, fine, pHeader\WObj:=wobj0;
		MoveL Openhole_690, v10, fine, pHeader\WObj:=wobj0;
		MoveL Openhole_691, v10, fine, pHeader\WObj:=wobj0;
		MoveL Openhole_692, v10, fine, pHeader\WObj:=wobj0;
		MoveL Openhole_693, v10, fine, pHeader\WObj:=wobj0;
		MoveL Openhole_694, v10, fine, pHeader\WObj:=wobj0;
		MoveL Openhole_695, v10, fine, pHeader\WObj:=wobj0;
		MoveL Openhole_696, v10, fine, pHeader\WObj:=wobj0;
		MoveL Openhole_697, v10, fine, pHeader\WObj:=wobj0;
		MoveL Openhole_698, v10, fine, pHeader\WObj:=wobj0;
		MoveL Openhole_699, v10, fine, pHeader\WObj:=wobj0;
		MoveL Openhole_700, v10, fine, pHeader\WObj:=wobj0;
		MoveL Openhole_701, v10, fine, pHeader\WObj:=wobj0;
		MoveL Openhole_702, v10, fine, pHeader\WObj:=wobj0;
		MoveL Openhole_703, v10, fine, pHeader\WObj:=wobj0;
		MoveL Openhole_704, v10, fine, pHeader\WObj:=wobj0;
		MoveL Openhole_705, v10, fine, pHeader\WObj:=wobj0;
		MoveL Openhole_706, v10, fine, pHeader\WObj:=wobj0;
		MoveL Openhole_707, v10, fine, pHeader\WObj:=wobj0;
		MoveL Openhole_708, v10, fine, pHeader\WObj:=wobj0;
		MoveL Openhole_709, v10, fine, pHeader\WObj:=wobj0;
		MoveL Openhole_710, v10, fine, pHeader\WObj:=wobj0;
		MoveL Openhole_711, v10, fine, pHeader\WObj:=wobj0;
		MoveL Openhole_712, v10, fine, pHeader\WObj:=wobj0;
		MoveL Openhole_713, v10, fine, pHeader\WObj:=wobj0;
		MoveL Openhole_714, v10, fine, pHeader\WObj:=wobj0;
		MoveL Openhole_715, v10, fine, pHeader\WObj:=wobj0;
		MoveL Openhole_716, v10, fine, pHeader\WObj:=wobj0;
		MoveL Openhole_717, v10, fine, pHeader\WObj:=wobj0;
		MoveL Openhole_718, v10, fine, pHeader\WObj:=wobj0;
		MoveL Openhole_719, v10, fine, pHeader\WObj:=wobj0;
		MoveL Openhole_720, v10, fine, pHeader\WObj:=wobj0;
		MoveL Openhole_721, v10, fine, pHeader\WObj:=wobj0;
		MoveL Openhole_722, v10, fine, pHeader\WObj:=wobj0;
		MoveL Openhole_723, v10, fine, pHeader\WObj:=wobj0;
		MoveL Openhole_724, v10, fine, pHeader\WObj:=wobj0;
		MoveL Openhole_725, v10, fine, pHeader\WObj:=wobj0;
		MoveL Openhole_726, v10, fine, pHeader\WObj:=wobj0;
		MoveL Openhole_727, v10, fine, pHeader\WObj:=wobj0;
		MoveL Openhole_728, v10, fine, pHeader\WObj:=wobj0;
		MoveL Openhole_729, v10, fine, pHeader\WObj:=wobj0;
		MoveL Openhole_730, v10, fine, pHeader\WObj:=wobj0;
		MoveL Openhole_731, v10, fine, pHeader\WObj:=wobj0;
		MoveL Openhole_732, v10, fine, pHeader\WObj:=wobj0;
		MoveL Openhole_733, v10, fine, pHeader\WObj:=wobj0;
		MoveL Openhole_734, v10, fine, pHeader\WObj:=wobj0;
		MoveL Openhole_735, v10, fine, pHeader\WObj:=wobj0;
		MoveL Openhole_736, v10, fine, pHeader\WObj:=wobj0;
		MoveL Openhole_737, v10, fine, pHeader\WObj:=wobj0;
		MoveL Openhole_738, v10, fine, pHeader\WObj:=wobj0;
		MoveL Openhole_739, v10, fine, pHeader\WObj:=wobj0;
		MoveL Openhole_740, v10, fine, pHeader\WObj:=wobj0;
		MoveL Openhole_741, v10, fine, pHeader\WObj:=wobj0;
		MoveL Openhole_742, v10, fine, pHeader\WObj:=wobj0;
		MoveL Openhole_743, v10, fine, pHeader\WObj:=wobj0;
		MoveL Openhole_744, v10, fine, pHeader\WObj:=wobj0;
		MoveL Openhole_745, v10, fine, pHeader\WObj:=wobj0;
		MoveL Openhole_746, v10, fine, pHeader\WObj:=wobj0;
		MoveL Openhole_747, v10, fine, pHeader\WObj:=wobj0;
		MoveL Openhole_748, v10, fine, pHeader\WObj:=wobj0;
		MoveL Openhole_749, v10, fine, pHeader\WObj:=wobj0;
		MoveL Openhole_750, v10, fine, pHeader\WObj:=wobj0;
		MoveL Openhole_751, v10, fine, pHeader\WObj:=wobj0;
		MoveL Openhole_752, v10, fine, pHeader\WObj:=wobj0;
		MoveL Openhole_753, v10, fine, pHeader\WObj:=wobj0;
		MoveL Openhole_754, v10, fine, pHeader\WObj:=wobj0;
		MoveL Openhole_755, v10, fine, pHeader\WObj:=wobj0;
		MoveL Openhole_756, v10, fine, pHeader\WObj:=wobj0;
		MoveL Openhole_757, v10, fine, pHeader\WObj:=wobj0;
		MoveL Openhole_758, v10, fine, pHeader\WObj:=wobj0;
		MoveL Openhole_759, v10, fine, pHeader\WObj:=wobj0;
		MoveL Openhole_760, v10, fine, pHeader\WObj:=wobj0;
		MoveL Openhole_761, v10, fine, pHeader\WObj:=wobj0;
		MoveL Openhole_762, v10, fine, pHeader\WObj:=wobj0;
		MoveL Openhole_763, v10, fine, pHeader\WObj:=wobj0;
		MoveL Openhole_764, v10, fine, pHeader\WObj:=wobj0;
		MoveL Openhole_765, v10, fine, pHeader\WObj:=wobj0;
		MoveL Openhole_766, v10, fine, pHeader\WObj:=wobj0;
		MoveL Openhole_767, v10, fine, pHeader\WObj:=wobj0;
		MoveL Openhole_768, v10, fine, pHeader\WObj:=wobj0;
		MoveL Openhole_769, v10, fine, pHeader\WObj:=wobj0;
		MoveL Openhole_770, v10, fine, pHeader\WObj:=wobj0;
		MoveL Openhole_771, v10, fine, pHeader\WObj:=wobj0;
		MoveL Openhole_772, v10, fine, pHeader\WObj:=wobj0;
		MoveL Openhole_773, v10, fine, pHeader\WObj:=wobj0;
		MoveL Openhole_774, v10, fine, pHeader\WObj:=wobj0;
		MoveL Openhole_775, v10, fine, pHeader\WObj:=wobj0;
		MoveL Openhole_776, v10, fine, pHeader\WObj:=wobj0;
		MoveL Openhole_777, v10, fine, pHeader\WObj:=wobj0;
		MoveL Openhole_778, v10, fine, pHeader\WObj:=wobj0;
		MoveL Openhole_779, v10, fine, pHeader\WObj:=wobj0;
		MoveL Openhole_780, v10, fine, pHeader\WObj:=wobj0;
		MoveL Openhole_781, v10, fine, pHeader\WObj:=wobj0;
		MoveL Openhole_782, v10, fine, pHeader\WObj:=wobj0;
		MoveL Openhole_783, v10, fine, pHeader\WObj:=wobj0;
		MoveL Openhole_784, v10, fine, pHeader\WObj:=wobj0;
		MoveL Openhole_785, v10, fine, pHeader\WObj:=wobj0;
		MoveL Openhole_786, v10, fine, pHeader\WObj:=wobj0;
		MoveL Openhole_787, v10, fine, pHeader\WObj:=wobj0;
		MoveL Openhole_788, v10, fine, pHeader\WObj:=wobj0;
		MoveL Openhole_789, v10, fine, pHeader\WObj:=wobj0;
		MoveL Openhole_790, v10, fine, pHeader\WObj:=wobj0;
		MoveL Openhole_791, v10, fine, pHeader\WObj:=wobj0;
		MoveL Openhole_792, v10, fine, pHeader\WObj:=wobj0;
		MoveL Openhole_793, v10, fine, pHeader\WObj:=wobj0;
		MoveL Openhole_794, v10, fine, pHeader\WObj:=wobj0;
		MoveL Openhole_795, v10, fine, pHeader\WObj:=wobj0;
		MoveL Openhole_796, v10, fine, pHeader\WObj:=wobj0;
		MoveL Openhole_797, v10, fine, pHeader\WObj:=wobj0;
		MoveL Openhole_798, v10, fine, pHeader\WObj:=wobj0;
		MoveL Openhole_799, v10, fine, pHeader\WObj:=wobj0;
		MoveL Openhole_800, v10, fine, pHeader\WObj:=wobj0;
		MoveL Openhole_801, v10, fine, pHeader\WObj:=wobj0;
		MoveL Openhole_802, v10, fine, pHeader\WObj:=wobj0;
		MoveL Openhole_803, v10, fine, pHeader\WObj:=wobj0;
		MoveL Openhole_804, v10, fine, pHeader\WObj:=wobj0;
		MoveL Openhole_805, v10, fine, pHeader\WObj:=wobj0;
		MoveL Openhole_806, v10, fine, pHeader\WObj:=wobj0;
		MoveL Openhole_807, v10, fine, pHeader\WObj:=wobj0;
		MoveL Openhole_808, v10, fine, pHeader\WObj:=wobj0;
		MoveL Openhole_809, v10, fine, pHeader\WObj:=wobj0;
		MoveL Openhole_810, v10, fine, pHeader\WObj:=wobj0;
		MoveL Openhole_811, v10, fine, pHeader\WObj:=wobj0;
		MoveL Openhole_812, v10, fine, pHeader\WObj:=wobj0;
		MoveL Openhole_813, v10, fine, pHeader\WObj:=wobj0;
		MoveL Openhole_814, v10, fine, pHeader\WObj:=wobj0;
		MoveL Openhole_815, v10, fine, pHeader\WObj:=wobj0;
		MoveL Openhole_816, v10, fine, pHeader\WObj:=wobj0;
		MoveL Openhole_817, v10, fine, pHeader\WObj:=wobj0;
		MoveL Openhole_818, v10, fine, pHeader\WObj:=wobj0;
		MoveL Openhole_819, v10, fine, pHeader\WObj:=wobj0;
		MoveL Openhole_820, v10, fine, pHeader\WObj:=wobj0;
		MoveL Openhole_821, v10, fine, pHeader\WObj:=wobj0;
		MoveL Openhole_822, v10, fine, pHeader\WObj:=wobj0;
		MoveL Openhole_823, v10, fine, pHeader\WObj:=wobj0;
		MoveL Openhole_824, v10, fine, pHeader\WObj:=wobj0;
		MoveL Openhole_825, v10, fine, pHeader\WObj:=wobj0;
		MoveL Openhole_826, v10, fine, pHeader\WObj:=wobj0;
		MoveL Openhole_827, v10, fine, pHeader\WObj:=wobj0;
		MoveL Openhole_828, v10, fine, pHeader\WObj:=wobj0;
		MoveL Openhole_829, v10, fine, pHeader\WObj:=wobj0;
		MoveL Openhole_830, v10, fine, pHeader\WObj:=wobj0;
		MoveL Openhole_831, v10, fine, pHeader\WObj:=wobj0;
		MoveL Openhole_832, v10, fine, pHeader\WObj:=wobj0;
		MoveL Openhole_833, v10, fine, pHeader\WObj:=wobj0;
		MoveL Openhole_834, v10, fine, pHeader\WObj:=wobj0;
		MoveL Openhole_835, v10, fine, pHeader\WObj:=wobj0;
		MoveL Openhole_836, v10, fine, pHeader\WObj:=wobj0;
		MoveL Openhole_837, v10, fine, pHeader\WObj:=wobj0;
		MoveL Openhole_838, v10, fine, pHeader\WObj:=wobj0;
		MoveL Openhole_839, v10, fine, pHeader\WObj:=wobj0;
		MoveL Openhole_840, v10, fine, pHeader\WObj:=wobj0;
		MoveL Openhole_841, v10, fine, pHeader\WObj:=wobj0;
		MoveL Openhole_842, v10, fine, pHeader\WObj:=wobj0;
		MoveL Openhole_843, v10, fine, pHeader\WObj:=wobj0;
		MoveL Openhole_844, v10, fine, pHeader\WObj:=wobj0;
		MoveL Openhole_845, v10, fine, pHeader\WObj:=wobj0;
		MoveL Openhole_846, v10, fine, pHeader\WObj:=wobj0;
		MoveL Openhole_847, v10, fine, pHeader\WObj:=wobj0;
		MoveL Openhole_848, v10, fine, pHeader\WObj:=wobj0;
		MoveL Openhole_849, v10, fine, pHeader\WObj:=wobj0;
		MoveL Openhole_850, v10, fine, pHeader\WObj:=wobj0;
		MoveL Openhole_851, v10, fine, pHeader\WObj:=wobj0;
		MoveL Openhole_852, v10, fine, pHeader\WObj:=wobj0;
		MoveL Openhole_853, v10, fine, pHeader\WObj:=wobj0;
		MoveL Openhole_854, v10, fine, pHeader\WObj:=wobj0;
		MoveL Openhole_855, v10, fine, pHeader\WObj:=wobj0;
		MoveL Openhole_856, v10, fine, pHeader\WObj:=wobj0;
		MoveL Openhole_857, v10, fine, pHeader\WObj:=wobj0;
		MoveL Openhole_858, v10, fine, pHeader\WObj:=wobj0;
		MoveL Openhole_859, v10, fine, pHeader\WObj:=wobj0;
		MoveL Openhole_860, v10, fine, pHeader\WObj:=wobj0;
		MoveL Openhole_861, v10, fine, pHeader\WObj:=wobj0;
		MoveL Openhole_862, v10, fine, pHeader\WObj:=wobj0;
		MoveL Openhole_863, v10, fine, pHeader\WObj:=wobj0;
		MoveL Openhole_864, v10, fine, pHeader\WObj:=wobj0;
		MoveL Openhole_865, v10, fine, pHeader\WObj:=wobj0;
		MoveL Openhole_866, v10, fine, pHeader\WObj:=wobj0;
		MoveL Openhole_867, v10, fine, pHeader\WObj:=wobj0;
		MoveL Openhole_868, v10, fine, pHeader\WObj:=wobj0;
		MoveL Openhole_869, v10, fine, pHeader\WObj:=wobj0;
		MoveL Openhole_870, v10, fine, pHeader\WObj:=wobj0;
		MoveL Openhole_871, v10, fine, pHeader\WObj:=wobj0;
		MoveL Openhole_872, v10, fine, pHeader\WObj:=wobj0;
		MoveL Openhole_873, v10, fine, pHeader\WObj:=wobj0;
		MoveL Openhole_874, v10, fine, pHeader\WObj:=wobj0;
		MoveL Openhole_875, v10, fine, pHeader\WObj:=wobj0;
		MoveL Openhole_876, v10, fine, pHeader\WObj:=wobj0;
		MoveL Openhole_877, v10, fine, pHeader\WObj:=wobj0;
		MoveL Openhole_878, v10, fine, pHeader\WObj:=wobj0;
		MoveL Openhole_879, v10, fine, pHeader\WObj:=wobj0;
		MoveL Openhole_880, v10, fine, pHeader\WObj:=wobj0;
		MoveL Openhole_881, v10, fine, pHeader\WObj:=wobj0;
		MoveL Openhole_882, v10, fine, pHeader\WObj:=wobj0;
		MoveL Openhole_883, v10, fine, pHeader\WObj:=wobj0;
		MoveL Openhole_884, v10, fine, pHeader\WObj:=wobj0;
		MoveL Openhole_885, v10, fine, pHeader\WObj:=wobj0;
		MoveL Openhole_886, v10, fine, pHeader\WObj:=wobj0;
		MoveL Openhole_887, v10, fine, pHeader\WObj:=wobj0;
		MoveL Openhole_888, v10, fine, pHeader\WObj:=wobj0;
		MoveL Openhole_889, v10, fine, pHeader\WObj:=wobj0;
		MoveL Openhole_890, v10, fine, pHeader\WObj:=wobj0;
		MoveL Openhole_891, v10, fine, pHeader\WObj:=wobj0;
		MoveL Openhole_892, v10, fine, pHeader\WObj:=wobj0;
		MoveL Openhole_893, v10, fine, pHeader\WObj:=wobj0;
		MoveL Openhole_894, v10, fine, pHeader\WObj:=wobj0;
		MoveL Openhole_895, v10, fine, pHeader\WObj:=wobj0;
		MoveL Openhole_896, v10, fine, pHeader\WObj:=wobj0;
		MoveL Openhole_897, v10, fine, pHeader\WObj:=wobj0;
		MoveL Openhole_898, v10, fine, pHeader\WObj:=wobj0;
		MoveL Openhole_899, v10, fine, pHeader\WObj:=wobj0;
		MoveL Openhole_900, v10, fine, pHeader\WObj:=wobj0;
		MoveL Openhole_901, v10, fine, pHeader\WObj:=wobj0;
		MoveL Openhole_902, v10, fine, pHeader\WObj:=wobj0;
		MoveL Openhole_903, v10, fine, pHeader\WObj:=wobj0;
		MoveL Openhole_904, v10, fine, pHeader\WObj:=wobj0;
		MoveL Openhole_905, v10, fine, pHeader\WObj:=wobj0;
		MoveL Openhole_906, v10, fine, pHeader\WObj:=wobj0;
		MoveL Openhole_907, v10, fine, pHeader\WObj:=wobj0;
		MoveL Openhole_908, v10, fine, pHeader\WObj:=wobj0;
		MoveL Openhole_909, v10, fine, pHeader\WObj:=wobj0;
		MoveL Openhole_910, v10, fine, pHeader\WObj:=wobj0;
		MoveL Openhole_911, v10, fine, pHeader\WObj:=wobj0;
		MoveL Openhole_912, v10, fine, pHeader\WObj:=wobj0;
		MoveL Openhole_913, v10, fine, pHeader\WObj:=wobj0;
		MoveL Openhole_914, v10, fine, pHeader\WObj:=wobj0;
		MoveL Openhole_915, v10, fine, pHeader\WObj:=wobj0;
		MoveL Openhole_916, v10, fine, pHeader\WObj:=wobj0;
		MoveL Openhole_917, v10, fine, pHeader\WObj:=wobj0;
		MoveL Openhole_918, v10, fine, pHeader\WObj:=wobj0;
		MoveL Openhole_919, v10, fine, pHeader\WObj:=wobj0;
		MoveL Openhole_920, v10, fine, pHeader\WObj:=wobj0;
		MoveL Openhole_921, v10, fine, pHeader\WObj:=wobj0;
		MoveL Openhole_922, v10, fine, pHeader\WObj:=wobj0;
		MoveL Openhole_923, v10, fine, pHeader\WObj:=wobj0;
		MoveL Openhole_924, v10, fine, pHeader\WObj:=wobj0;
		MoveL Openhole_925, v10, fine, pHeader\WObj:=wobj0;
		MoveL Openhole_926, v10, fine, pHeader\WObj:=wobj0;
		MoveL Openhole_927, v10, fine, pHeader\WObj:=wobj0;
		MoveL Openhole_928, v10, fine, pHeader\WObj:=wobj0;
		MoveL Openhole_929, v10, fine, pHeader\WObj:=wobj0;
		MoveL Openhole_930, v10, fine, pHeader\WObj:=wobj0;
		MoveL Openhole_931, v10, fine, pHeader\WObj:=wobj0;
		MoveL Openhole_932, v10, fine, pHeader\WObj:=wobj0;
		MoveL Openhole_933, v10, fine, pHeader\WObj:=wobj0;
		MoveL Openhole_934, v10, fine, pHeader\WObj:=wobj0;
		MoveL Openhole_935, v10, fine, pHeader\WObj:=wobj0;
		MoveL Openhole_936, v10, fine, pHeader\WObj:=wobj0;
		MoveL Openhole_937, v10, fine, pHeader\WObj:=wobj0;
		MoveL Openhole_938, v10, fine, pHeader\WObj:=wobj0;
		MoveL Openhole_939, v10, fine, pHeader\WObj:=wobj0;
		MoveL Openhole_940, v10, fine, pHeader\WObj:=wobj0;
		MoveL Openhole_941, v10, fine, pHeader\WObj:=wobj0;
		MoveL Openhole_942, v10, fine, pHeader\WObj:=wobj0;
		MoveL Openhole_943, v10, fine, pHeader\WObj:=wobj0;
		MoveL Openhole_944, v10, fine, pHeader\WObj:=wobj0;
		MoveL Openhole_945, v10, fine, pHeader\WObj:=wobj0;
		MoveL Openhole_946, v10, fine, pHeader\WObj:=wobj0;
		MoveL Openhole_947, v10, fine, pHeader\WObj:=wobj0;
		MoveL Openhole_948, v10, fine, pHeader\WObj:=wobj0;
		MoveL Openhole_949, v10, fine, pHeader\WObj:=wobj0;
		MoveL Openhole_950, v10, fine, pHeader\WObj:=wobj0;
		MoveL Openhole_951, v10, fine, pHeader\WObj:=wobj0;
		MoveL Openhole_952, v10, fine, pHeader\WObj:=wobj0;
		MoveL Openhole_953, v10, fine, pHeader\WObj:=wobj0;
		MoveL Openhole_954, v10, fine, pHeader\WObj:=wobj0;
		MoveL Openhole_955, v10, fine, pHeader\WObj:=wobj0;
		MoveL Openhole_956, v10, fine, pHeader\WObj:=wobj0;
		MoveL Openhole_957, v10, fine, pHeader\WObj:=wobj0;
		MoveL Openhole_958, v10, fine, pHeader\WObj:=wobj0;
		MoveL Openhole_959, v10, fine, pHeader\WObj:=wobj0;
		MoveL Openhole_960, v10, fine, pHeader\WObj:=wobj0;
		MoveL Openhole_961, v10, fine, pHeader\WObj:=wobj0;
		MoveL Openhole_962, v10, fine, pHeader\WObj:=wobj0;
		MoveL Openhole_963, v10, fine, pHeader\WObj:=wobj0;
		MoveL Openhole_964, v10, fine, pHeader\WObj:=wobj0;
		MoveL Openhole_965, v10, fine, pHeader\WObj:=wobj0;
		MoveL Openhole_966, v10, fine, pHeader\WObj:=wobj0;
		MoveL Openhole_967, v10, fine, pHeader\WObj:=wobj0;
		MoveL Openhole_968, v10, fine, pHeader\WObj:=wobj0;
		MoveL Openhole_969, v10, fine, pHeader\WObj:=wobj0;
		MoveL Openhole_970, v10, fine, pHeader\WObj:=wobj0;
		MoveL Openhole_971, v10, fine, pHeader\WObj:=wobj0;
		MoveL Openhole_972, v10, fine, pHeader\WObj:=wobj0;
		MoveL Openhole_973, v10, fine, pHeader\WObj:=wobj0;
		MoveL Openhole_974, v10, fine, pHeader\WObj:=wobj0;
		MoveL Openhole_975, v10, fine, pHeader\WObj:=wobj0;
		MoveL Openhole_976, v10, fine, pHeader\WObj:=wobj0;
		MoveL Openhole_977, v10, fine, pHeader\WObj:=wobj0;
		MoveL Openhole_978, v10, fine, pHeader\WObj:=wobj0;
		MoveL Openhole_979, v10, fine, pHeader\WObj:=wobj0;
		MoveL Openhole_980, v10, fine, pHeader\WObj:=wobj0;
		MoveL Openhole_981, v10, fine, pHeader\WObj:=wobj0;
		MoveL Openhole_982, v10, fine, pHeader\WObj:=wobj0;
		MoveL Openhole_983, v10, fine, pHeader\WObj:=wobj0;
		MoveL Openhole_984, v10, fine, pHeader\WObj:=wobj0;
		MoveL Openhole_985, v10, fine, pHeader\WObj:=wobj0;
		MoveL Openhole_986, v10, fine, pHeader\WObj:=wobj0;
		MoveL Openhole_987, v10, fine, pHeader\WObj:=wobj0;
		MoveL Openhole_988, v10, fine, pHeader\WObj:=wobj0;
		MoveL Openhole_989, v10, fine, pHeader\WObj:=wobj0;
		MoveL Openhole_990, v10, fine, pHeader\WObj:=wobj0;
		MoveL Openhole_991, v10, fine, pHeader\WObj:=wobj0;
		MoveL Openhole_992, v10, fine, pHeader\WObj:=wobj0;
		MoveL Openhole_993, v10, fine, pHeader\WObj:=wobj0;
		MoveL Openhole_994, v10, fine, pHeader\WObj:=wobj0;
		MoveL Openhole_995, v10, fine, pHeader\WObj:=wobj0;
		MoveL Openhole_996, v10, fine, pHeader\WObj:=wobj0;
		MoveL Openhole_997, v10, fine, pHeader\WObj:=wobj0;
		MoveL Openhole_998, v10, fine, pHeader\WObj:=wobj0;
		MoveL Openhole_999, v10, fine, pHeader\WObj:=wobj0;
		MoveL Openhole_1000, v10, fine, pHeader\WObj:=wobj0;
		MoveL Openhole_1001, v10, fine, pHeader\WObj:=wobj0;
		MoveL Openhole_1002, v10, fine, pHeader\WObj:=wobj0;
		MoveL Openhole_1003, v10, fine, pHeader\WObj:=wobj0;
		MoveL Openhole_1004, v10, fine, pHeader\WObj:=wobj0;
		MoveL Openhole_1005, v10, fine, pHeader\WObj:=wobj0;
		MoveL Openhole_1006, v10, fine, pHeader\WObj:=wobj0;
		MoveL Openhole_1007, v10, fine, pHeader\WObj:=wobj0;
		MoveL Openhole_1008, v10, fine, pHeader\WObj:=wobj0;
		MoveL Openhole_1009, v10, fine, pHeader\WObj:=wobj0;
		MoveL Openhole_1010, v10, fine, pHeader\WObj:=wobj0;
		MoveL Openhole_1011, v10, fine, pHeader\WObj:=wobj0;
		MoveL Openhole_1012, v10, fine, pHeader\WObj:=wobj0;
		MoveL Openhole_1013, v10, fine, pHeader\WObj:=wobj0;
		MoveL Openhole_1014, v10, fine, pHeader\WObj:=wobj0;
		MoveL Openhole_1015, v10, fine, pHeader\WObj:=wobj0;
		MoveL Openhole_1016, v10, fine, pHeader\WObj:=wobj0;
		MoveL Openhole_1017, v10, fine, pHeader\WObj:=wobj0;
		MoveL Openhole_1018, v10, fine, pHeader\WObj:=wobj0;
		MoveL Openhole_1019, v10, fine, pHeader\WObj:=wobj0;
		MoveL Openhole_1020, v10, fine, pHeader\WObj:=wobj0;
		MoveL Openhole_1021, v10, fine, pHeader\WObj:=wobj0;
		MoveL Openhole_1022, v10, fine, pHeader\WObj:=wobj0;
		MoveL Openhole_1023, v10, fine, pHeader\WObj:=wobj0;
		MoveL Openhole_1024, v10, fine, pHeader\WObj:=wobj0;
		MoveL Openhole_1025, v10, fine, pHeader\WObj:=wobj0;
		MoveL Openhole_1026, v10, fine, pHeader\WObj:=wobj0;
		MoveL Openhole_1027, v10, fine, pHeader\WObj:=wobj0;
		MoveL Openhole_1028, v10, fine, pHeader\WObj:=wobj0;
		MoveL Openhole_1029, v10, fine, pHeader\WObj:=wobj0;
		MoveL Openhole_1030, v10, fine, pHeader\WObj:=wobj0;
		MoveL Openhole_1031, v10, fine, pHeader\WObj:=wobj0;
		MoveL Openhole_1032, v10, fine, pHeader\WObj:=wobj0;
		MoveL Openhole_1033, v10, fine, pHeader\WObj:=wobj0;
		MoveL Openhole_1034, v10, fine, pHeader\WObj:=wobj0;
		MoveL Openhole_1035, v10, fine, pHeader\WObj:=wobj0;
		MoveL Openhole_1036, v10, fine, pHeader\WObj:=wobj0;
		MoveL Openhole_1037, v10, fine, pHeader\WObj:=wobj0;
		MoveL Openhole_1038, v10, fine, pHeader\WObj:=wobj0;
		MoveL Openhole_1039, v10, fine, pHeader\WObj:=wobj0;
		MoveL Openhole_1040, v10, fine, pHeader\WObj:=wobj0;
		MoveL Openhole_1041, v10, fine, pHeader\WObj:=wobj0;
		MoveL Openhole_1042, v10, fine, pHeader\WObj:=wobj0;
		MoveL Openhole_1043, v10, fine, pHeader\WObj:=wobj0;
		MoveL Openhole_1044, v10, fine, pHeader\WObj:=wobj0;
		MoveL Openhole_1045, v10, fine, pHeader\WObj:=wobj0;
		MoveL Openhole_1046, v10, fine, pHeader\WObj:=wobj0;
		MoveL Openhole_1047, v10, fine, pHeader\WObj:=wobj0;
		MoveL Openhole_1048, v10, fine, pHeader\WObj:=wobj0;
		MoveL Openhole_1049, v10, fine, pHeader\WObj:=wobj0;
		MoveL Openhole_1050, v10, fine, pHeader\WObj:=wobj0;
		MoveL Openhole_1051, v10, fine, pHeader\WObj:=wobj0;
		MoveL Openhole_1052, v10, fine, pHeader\WObj:=wobj0;
		MoveL Openhole_1053, v10, fine, pHeader\WObj:=wobj0;
		MoveL Openhole_1054, v10, fine, pHeader\WObj:=wobj0;
		MoveL Openhole_1055, v10, fine, pHeader\WObj:=wobj0;
		MoveL Openhole_1056, v10, fine, pHeader\WObj:=wobj0;
		MoveL Openhole_1057, v10, fine, pHeader\WObj:=wobj0;
		MoveL Openhole_1058, v10, fine, pHeader\WObj:=wobj0;
		MoveL Openhole_1059, v10, fine, pHeader\WObj:=wobj0;
		MoveL Openhole_1060, v10, fine, pHeader\WObj:=wobj0;
		MoveL Openhole_1061, v10, fine, pHeader\WObj:=wobj0;
		MoveL Openhole_1062, v10, fine, pHeader\WObj:=wobj0;
		MoveL Openhole_1063, v10, fine, pHeader\WObj:=wobj0;
		MoveL Openhole_1064, v10, fine, pHeader\WObj:=wobj0;
		MoveL Openhole_1065, v10, fine, pHeader\WObj:=wobj0;
		MoveL Openhole_1066, v10, fine, pHeader\WObj:=wobj0;
		MoveL Openhole_1067, v10, fine, pHeader\WObj:=wobj0;
		MoveL Openhole_1068, v10, fine, pHeader\WObj:=wobj0;
		MoveL Openhole_1069, v10, fine, pHeader\WObj:=wobj0;
		MoveL Openhole_1070, v10, fine, pHeader\WObj:=wobj0;
		MoveL Openhole_1071, v10, fine, pHeader\WObj:=wobj0;
		MoveL Openhole_1072, v10, fine, pHeader\WObj:=wobj0;
		MoveL Openhole_1073, v10, fine, pHeader\WObj:=wobj0;
		MoveL Openhole_1074, v10, fine, pHeader\WObj:=wobj0;
		MoveL Openhole_1075, v10, fine, pHeader\WObj:=wobj0;
		MoveL Openhole_1076, v10, fine, pHeader\WObj:=wobj0;
		MoveL Openhole_1077, v10, fine, pHeader\WObj:=wobj0;
		MoveL Openhole_1078, v10, fine, pHeader\WObj:=wobj0;
		MoveL Openhole_1079, v10, fine, pHeader\WObj:=wobj0;
		MoveL Openhole_1080, v10, fine, pHeader\WObj:=wobj0;
		MoveL Openhole_1081, v10, fine, pHeader\WObj:=wobj0;
		MoveL Openhole_1082, v10, fine, pHeader\WObj:=wobj0;
		MoveL Openhole_1083, v10, fine, pHeader\WObj:=wobj0;
		MoveL Openhole_1084, v10, fine, pHeader\WObj:=wobj0;
		MoveL Openhole_1085, v10, fine, pHeader\WObj:=wobj0;
		MoveL Openhole_1086, v10, fine, pHeader\WObj:=wobj0;
		MoveL Openhole_1087, v10, fine, pHeader\WObj:=wobj0;
		MoveL Openhole_1088, v10, fine, pHeader\WObj:=wobj0;
		MoveL Openhole_1089, v10, fine, pHeader\WObj:=wobj0;
		MoveL Openhole_1090, v10, fine, pHeader\WObj:=wobj0;
		MoveL Openhole_1091, v10, fine, pHeader\WObj:=wobj0;
		MoveL Openhole_1092, v10, fine, pHeader\WObj:=wobj0;
		MoveL Openhole_1093, v10, fine, pHeader\WObj:=wobj0;
		MoveL Openhole_1094, v10, fine, pHeader\WObj:=wobj0;
		MoveL Openhole_1095, v10, fine, pHeader\WObj:=wobj0;
		MoveL Openhole_1096, v10, fine, pHeader\WObj:=wobj0;
		MoveL Openhole_1097, v10, fine, pHeader\WObj:=wobj0;
		MoveL Openhole_1098, v10, fine, pHeader\WObj:=wobj0;
		MoveL Openhole_1099, v10, fine, pHeader\WObj:=wobj0;
		MoveL Openhole_1100, v10, fine, pHeader\WObj:=wobj0;
		MoveL Openhole_1101, v10, fine, pHeader\WObj:=wobj0;
		MoveL Openhole_1102, v10, fine, pHeader\WObj:=wobj0;
		MoveL Openhole_1103, v10, fine, pHeader\WObj:=wobj0;
		MoveL Openhole_1104, v10, fine, pHeader\WObj:=wobj0;
		MoveL Openhole_1105, v10, fine, pHeader\WObj:=wobj0;
		MoveL Openhole_1106, v10, fine, pHeader\WObj:=wobj0;
		MoveL Openhole_1107, v10, fine, pHeader\WObj:=wobj0;
		MoveL Openhole_1108, v10, fine, pHeader\WObj:=wobj0;
		MoveL Openhole_1109, v10, fine, pHeader\WObj:=wobj0;
		MoveL Openhole_1110, v10, fine, pHeader\WObj:=wobj0;
		MoveL Openhole_1111, v10, fine, pHeader\WObj:=wobj0;
		MoveL Openhole_1112, v10, fine, pHeader\WObj:=wobj0;
		MoveL Openhole_1113, v10, fine, pHeader\WObj:=wobj0;
		MoveL Openhole_1114, v10, fine, pHeader\WObj:=wobj0;
		MoveL Openhole_1115, v10, fine, pHeader\WObj:=wobj0;
		MoveL Openhole_1116, v10, fine, pHeader\WObj:=wobj0;
		MoveL Openhole_1117, v10, fine, pHeader\WObj:=wobj0;
		MoveL Openhole_1118, v10, fine, pHeader\WObj:=wobj0;
		MoveL Openhole_1119, v10, fine, pHeader\WObj:=wobj0;
		MoveL Openhole_1120, v10, fine, pHeader\WObj:=wobj0;
		MoveL Openhole_1121, v10, fine, pHeader\WObj:=wobj0;
		MoveL Openhole_1122, v10, fine, pHeader\WObj:=wobj0;
		MoveL Openhole_1123, v10, fine, pHeader\WObj:=wobj0;
		MoveL Openhole_1124, v10, fine, pHeader\WObj:=wobj0;
		MoveL Openhole_1125, v10, fine, pHeader\WObj:=wobj0;
		MoveL Openhole_1126, v10, fine, pHeader\WObj:=wobj0;
		MoveL Openhole_1127, v10, fine, pHeader\WObj:=wobj0;
		MoveL Openhole_1128, v10, fine, pHeader\WObj:=wobj0;
		MoveL Openhole_1129, v10, fine, pHeader\WObj:=wobj0;
		MoveL Openhole_1130, v10, fine, pHeader\WObj:=wobj0;
		MoveL Openhole_1131, v10, fine, pHeader\WObj:=wobj0;
		MoveL Openhole_1132, v10, fine, pHeader\WObj:=wobj0;
		MoveL Openhole_1133, v10, fine, pHeader\WObj:=wobj0;
		MoveL Openhole_1134, v10, fine, pHeader\WObj:=wobj0;
		MoveL Openhole_1135, v10, fine, pHeader\WObj:=wobj0;
		MoveL Openhole_1136, v10, fine, pHeader\WObj:=wobj0;
		MoveL Openhole_1137, v10, fine, pHeader\WObj:=wobj0;
		MoveL Openhole_1138, v10, fine, pHeader\WObj:=wobj0;
		MoveL Openhole_1139, v10, fine, pHeader\WObj:=wobj0;
		MoveL Openhole_1140, v10, fine, pHeader\WObj:=wobj0;
		MoveL Openhole_1141, v10, fine, pHeader\WObj:=wobj0;
		MoveL Openhole_1142, v10, fine, pHeader\WObj:=wobj0;
		MoveL Openhole_1143, v10, fine, pHeader\WObj:=wobj0;
		MoveL Openhole_1144, v10, fine, pHeader\WObj:=wobj0;
		MoveL Openhole_1145, v10, fine, pHeader\WObj:=wobj0;
		MoveL Openhole_1146, v10, fine, pHeader\WObj:=wobj0;
		MoveL Openhole_1147, v10, fine, pHeader\WObj:=wobj0;
		MoveL Openhole_1148, v10, fine, pHeader\WObj:=wobj0;
		MoveL Openhole_1149, v10, fine, pHeader\WObj:=wobj0;
		MoveL Openhole_1150, v10, fine, pHeader\WObj:=wobj0;
		MoveL Openhole_1151, v10, fine, pHeader\WObj:=wobj0;
		MoveL Openhole_1152, v10, fine, pHeader\WObj:=wobj0;
		MoveL Openhole_1153, v10, fine, pHeader\WObj:=wobj0;
		MoveL Openhole_1154, v10, fine, pHeader\WObj:=wobj0;
		MoveL Openhole_1155, v10, fine, pHeader\WObj:=wobj0;
		MoveL Openhole_1156, v10, fine, pHeader\WObj:=wobj0;
		MoveL Openhole_1157, v10, fine, pHeader\WObj:=wobj0;
		MoveL Openhole_1158, v10, fine, pHeader\WObj:=wobj0;
		MoveL Openhole_1159, v10, fine, pHeader\WObj:=wobj0;
		MoveL Openhole_1160, v10, fine, pHeader\WObj:=wobj0;
		MoveL Openhole_1161, v10, fine, pHeader\WObj:=wobj0;
		MoveL Openhole_1162, v10, fine, pHeader\WObj:=wobj0;
		MoveL Openhole_1163, v10, fine, pHeader\WObj:=wobj0;
		MoveL Openhole_1164, v10, fine, pHeader\WObj:=wobj0;
		MoveL Openhole_1165, v10, fine, pHeader\WObj:=wobj0;
		MoveL Openhole_1166, v10, fine, pHeader\WObj:=wobj0;
		MoveL Openhole_1167, v10, fine, pHeader\WObj:=wobj0;
		MoveL Openhole_1168, v10, fine, pHeader\WObj:=wobj0;
		MoveL Openhole_1169, v10, fine, pHeader\WObj:=wobj0;
		MoveL Openhole_1170, v10, fine, pHeader\WObj:=wobj0;
		MoveL Openhole_1171, v10, fine, pHeader\WObj:=wobj0;
		MoveL Openhole_1172, v10, fine, pHeader\WObj:=wobj0;
		MoveL Openhole_1173, v10, fine, pHeader\WObj:=wobj0;
		MoveL Openhole_1174, v10, fine, pHeader\WObj:=wobj0;
		MoveL Openhole_1175, v10, fine, pHeader\WObj:=wobj0;
		MoveL Openhole_1176, v10, fine, pHeader\WObj:=wobj0;
		MoveL Openhole_1177, v10, fine, pHeader\WObj:=wobj0;
		MoveL Openhole_1178, v10, fine, pHeader\WObj:=wobj0;
		MoveL Openhole_1179, v10, fine, pHeader\WObj:=wobj0;
		MoveL Openhole_1180, v10, fine, pHeader\WObj:=wobj0;
		MoveL Openhole_1181, v10, fine, pHeader\WObj:=wobj0;
		MoveL Openhole_1182, v10, fine, pHeader\WObj:=wobj0;
		MoveL Openhole_1183, v10, fine, pHeader\WObj:=wobj0;
		MoveL Openhole_1184, v10, fine, pHeader\WObj:=wobj0;
		MoveL Openhole_1185, v10, fine, pHeader\WObj:=wobj0;
		MoveL Openhole_1186, v10, fine, pHeader\WObj:=wobj0;
		MoveL Openhole_1187, v10, fine, pHeader\WObj:=wobj0;
		MoveL Openhole_1188, v10, fine, pHeader\WObj:=wobj0;
		MoveL Openhole_1189, v10, fine, pHeader\WObj:=wobj0;
		MoveL Openhole_1190, v10, fine, pHeader\WObj:=wobj0;
		MoveL Openhole_1191, v10, fine, pHeader\WObj:=wobj0;
		MoveL Openhole_1192, v10, fine, pHeader\WObj:=wobj0;
		MoveL Openhole_1193, v10, fine, pHeader\WObj:=wobj0;
		MoveL Openhole_1194, v10, fine, pHeader\WObj:=wobj0;
		MoveL Openhole_1195, v10, fine, pHeader\WObj:=wobj0;
		MoveL Openhole_1196, v10, fine, pHeader\WObj:=wobj0;
		MoveL Openhole_1197, v10, fine, pHeader\WObj:=wobj0;
		MoveL Openhole_1198, v10, fine, pHeader\WObj:=wobj0;
		MoveL Openhole_1199, v10, fine, pHeader\WObj:=wobj0;
		MoveL Openhole_1200, v10, fine, pHeader\WObj:=wobj0;
		MoveL Openhole_1201, v10, fine, pHeader\WObj:=wobj0;
		MoveL Openhole_1202, v10, fine, pHeader\WObj:=wobj0;
		MoveL Openhole_1203, v10, fine, pHeader\WObj:=wobj0;
		MoveL Openhole_1204, v10, fine, pHeader\WObj:=wobj0;
		MoveL Openhole_1205, v10, fine, pHeader\WObj:=wobj0;
		MoveL Openhole_1206, v10, fine, pHeader\WObj:=wobj0;
		MoveL Openhole_1207, v10, fine, pHeader\WObj:=wobj0;
		MoveL Openhole_1208, v10, fine, pHeader\WObj:=wobj0;
		MoveL Openhole_1209, v10, fine, pHeader\WObj:=wobj0;
		MoveL Openhole_1210, v10, fine, pHeader\WObj:=wobj0;
		MoveL Openhole_1211, v10, fine, pHeader\WObj:=wobj0;
		MoveL Openhole_1212, v10, fine, pHeader\WObj:=wobj0;
		MoveL Openhole_1213, v10, fine, pHeader\WObj:=wobj0;
		MoveL Openhole_1214, v10, fine, pHeader\WObj:=wobj0;
		MoveL Openhole_1215, v10, fine, pHeader\WObj:=wobj0;
		MoveL Openhole_1216, v10, fine, pHeader\WObj:=wobj0;
		MoveL Openhole_1217, v10, fine, pHeader\WObj:=wobj0;
		MoveL Openhole_1218, v10, fine, pHeader\WObj:=wobj0;
		MoveL Openhole_1219, v10, fine, pHeader\WObj:=wobj0;
		MoveL Openhole_1220, v10, fine, pHeader\WObj:=wobj0;
		MoveL Openhole_1221, v10, fine, pHeader\WObj:=wobj0;
		MoveL Openhole_1222, v10, fine, pHeader\WObj:=wobj0;
		MoveL Openhole_1223, v10, fine, pHeader\WObj:=wobj0;
		MoveL Openhole_1224, v10, fine, pHeader\WObj:=wobj0;
		MoveL Openhole_1225, v10, fine, pHeader\WObj:=wobj0;
		MoveL Openhole_1226, v10, fine, pHeader\WObj:=wobj0;
		MoveL Openhole_1227, v10, fine, pHeader\WObj:=wobj0;
		MoveL Openhole_1228, v10, fine, pHeader\WObj:=wobj0;
		MoveL Openhole_1229, v10, fine, pHeader\WObj:=wobj0;
		MoveL Openhole_1230, v10, fine, pHeader\WObj:=wobj0;
		MoveL Openhole_1231, v10, fine, pHeader\WObj:=wobj0;
		MoveL Openhole_1232, v10, fine, pHeader\WObj:=wobj0;
		MoveL Openhole_1233, v10, fine, pHeader\WObj:=wobj0;
		MoveL Openhole_1234, v10, fine, pHeader\WObj:=wobj0;
		MoveL Openhole_1235, v10, fine, pHeader\WObj:=wobj0;
		MoveL Openhole_1236, v10, fine, pHeader\WObj:=wobj0;
		MoveL Openhole_1237, v10, fine, pHeader\WObj:=wobj0;
		MoveL Openhole_1238, v10, fine, pHeader\WObj:=wobj0;
		MoveL Openhole_1239, v10, fine, pHeader\WObj:=wobj0;
		MoveL Openhole_1240, v10, fine, pHeader\WObj:=wobj0;
		MoveL Openhole_1241, v10, fine, pHeader\WObj:=wobj0;
		MoveL Openhole_1242, v10, fine, pHeader\WObj:=wobj0;
		MoveL Openhole_1243, v10, fine, pHeader\WObj:=wobj0;
		MoveL Openhole_1244, v10, fine, pHeader\WObj:=wobj0;
		MoveL Openhole_1245, v10, fine, pHeader\WObj:=wobj0;
		MoveL Openhole_1246, v10, fine, pHeader\WObj:=wobj0;
		MoveL Openhole_1247, v10, fine, pHeader\WObj:=wobj0;
		MoveL Openhole_1248, v10, fine, pHeader\WObj:=wobj0;
		MoveL Openhole_1249, v10, fine, pHeader\WObj:=wobj0;
		MoveL Openhole_1250, v10, fine, pHeader\WObj:=wobj0;
		MoveL Openhole_1251, v10, fine, pHeader\WObj:=wobj0;
		MoveL Openhole_1252, v10, fine, pHeader\WObj:=wobj0;
		MoveL Openhole_1253, v10, fine, pHeader\WObj:=wobj0;
		MoveL Openhole_1254, v10, fine, pHeader\WObj:=wobj0;
		MoveL Openhole_1255, v10, fine, pHeader\WObj:=wobj0;
		MoveL Openhole_1256, v10, fine, pHeader\WObj:=wobj0;
		MoveL Openhole_1257, v10, fine, pHeader\WObj:=wobj0;
		MoveL Openhole_1258, v10, fine, pHeader\WObj:=wobj0;
		MoveL Openhole_1259, v10, fine, pHeader\WObj:=wobj0;
		MoveL Openhole_1260, v10, fine, pHeader\WObj:=wobj0;
		MoveL Openhole_1261, v10, fine, pHeader\WObj:=wobj0;
		MoveL Openhole_1262, v10, fine, pHeader\WObj:=wobj0;
		MoveL Openhole_1263, v10, fine, pHeader\WObj:=wobj0;
		MoveL Openhole_1264, v10, fine, pHeader\WObj:=wobj0;
		MoveL Openhole_1265, v10, fine, pHeader\WObj:=wobj0;
		MoveL Openhole_1266, v10, fine, pHeader\WObj:=wobj0;
		MoveL Openhole_1267, v10, fine, pHeader\WObj:=wobj0;
		MoveL Openhole_1268, v10, fine, pHeader\WObj:=wobj0;
		MoveL Openhole_1269, v10, fine, pHeader\WObj:=wobj0;
		MoveL Openhole_1270, v10, fine, pHeader\WObj:=wobj0;
		MoveL Openhole_1271, v10, fine, pHeader\WObj:=wobj0;
		MoveL Openhole_1272, v10, fine, pHeader\WObj:=wobj0;
		MoveL Openhole_1273, v10, fine, pHeader\WObj:=wobj0;
		MoveL Openhole_1274, v10, fine, pHeader\WObj:=wobj0;
		MoveL Openhole_1275, v10, fine, pHeader\WObj:=wobj0;
		MoveL Openhole_1276, v10, fine, pHeader\WObj:=wobj0;
		MoveL Openhole_1277, v10, fine, pHeader\WObj:=wobj0;
		MoveL Openhole_1278, v10, fine, pHeader\WObj:=wobj0;
		MoveL Openhole_1279, v10, fine, pHeader\WObj:=wobj0;
		MoveL Openhole_1280, v10, fine, pHeader\WObj:=wobj0;
		MoveL Openhole_1281, v10, fine, pHeader\WObj:=wobj0;
		MoveL Openhole_1282, v10, fine, pHeader\WObj:=wobj0;
		MoveL Openhole_1283, v10, fine, pHeader\WObj:=wobj0;
		MoveL Openhole_1284, v10, fine, pHeader\WObj:=wobj0;
		MoveL Openhole_1285, v10, fine, pHeader\WObj:=wobj0;
		MoveL Openhole_1286, v10, fine, pHeader\WObj:=wobj0;
		MoveL Openhole_1287, v10, fine, pHeader\WObj:=wobj0;
		MoveL Openhole_1288, v10, fine, pHeader\WObj:=wobj0;
		MoveL Openhole_1289, v10, fine, pHeader\WObj:=wobj0;
		MoveL Openhole_1290, v10, fine, pHeader\WObj:=wobj0;
		MoveL Openhole_1291, v10, fine, pHeader\WObj:=wobj0;
		MoveL Openhole_1292, v10, fine, pHeader\WObj:=wobj0;
		MoveL Openhole_1293, v10, fine, pHeader\WObj:=wobj0;
		MoveL Openhole_1294, v10, fine, pHeader\WObj:=wobj0;
		MoveL Openhole_1295, v10, fine, pHeader\WObj:=wobj0;
		MoveL Openhole_1296, v10, fine, pHeader\WObj:=wobj0;
		MoveL Openhole_1297, v10, fine, pHeader\WObj:=wobj0;
		MoveL Openhole_1298, v10, fine, pHeader\WObj:=wobj0;
		MoveL Openhole_1299, v10, fine, pHeader\WObj:=wobj0;
		MoveL Openhole_1300, v10, fine, pHeader\WObj:=wobj0;
		MoveL Openhole_1301, v10, fine, pHeader\WObj:=wobj0;
		MoveL Openhole_1302, v10, fine, pHeader\WObj:=wobj0;
		MoveL Openhole_1303, v10, fine, pHeader\WObj:=wobj0;
		MoveL Openhole_1304, v10, fine, pHeader\WObj:=wobj0;
		MoveL Openhole_1305, v10, fine, pHeader\WObj:=wobj0;
		MoveL Openhole_1306, v10, fine, pHeader\WObj:=wobj0;
		MoveL Openhole_1307, v10, fine, pHeader\WObj:=wobj0;
		MoveL Openhole_1308, v10, fine, pHeader\WObj:=wobj0;
		MoveL Openhole_1309, v10, fine, pHeader\WObj:=wobj0;
		MoveL Openhole_1310, v10, fine, pHeader\WObj:=wobj0;
		MoveL Openhole_1311, v10, fine, pHeader\WObj:=wobj0;
		MoveL Openhole_1312, v10, fine, pHeader\WObj:=wobj0;
		MoveL Openhole_1313, v10, fine, pHeader\WObj:=wobj0;
		MoveL Openhole_1314, v10, fine, pHeader\WObj:=wobj0;
		MoveL Openhole_1315, v10, fine, pHeader\WObj:=wobj0;
		MoveL Openhole_1316, v10, fine, pHeader\WObj:=wobj0;
		MoveL Openhole_1317, v10, fine, pHeader\WObj:=wobj0;
		MoveL Openhole_1318, v10, fine, pHeader\WObj:=wobj0;
		MoveL Openhole_1319, v10, fine, pHeader\WObj:=wobj0;
		MoveL Openhole_1320, v10, fine, pHeader\WObj:=wobj0;
		MoveL Openhole_1321, v10, fine, pHeader\WObj:=wobj0;
		MoveL Openhole_1322, v10, fine, pHeader\WObj:=wobj0;
		MoveL Openhole_1323, v10, fine, pHeader\WObj:=wobj0;
		MoveL Openhole_1324, v10, fine, pHeader\WObj:=wobj0;
		MoveL Openhole_1325, v10, fine, pHeader\WObj:=wobj0;
		MoveL Openhole_1326, v10, fine, pHeader\WObj:=wobj0;
		MoveL Openhole_1327, v10, fine, pHeader\WObj:=wobj0;
		MoveL Openhole_1328, v10, fine, pHeader\WObj:=wobj0;
		MoveL Openhole_1329, v10, fine, pHeader\WObj:=wobj0;
		MoveL Openhole_1330, v10, fine, pHeader\WObj:=wobj0;
		MoveL Openhole_1331, v10, fine, pHeader\WObj:=wobj0;
		MoveL Openhole_1332, v10, fine, pHeader\WObj:=wobj0;
		MoveL Openhole_1333, v10, fine, pHeader\WObj:=wobj0;
		MoveL Openhole_1334, v10, fine, pHeader\WObj:=wobj0;
		MoveL Openhole_1335, v10, fine, pHeader\WObj:=wobj0;
		MoveL Openhole_1336, v10, fine, pHeader\WObj:=wobj0;
		MoveL Openhole_1337, v10, fine, pHeader\WObj:=wobj0;
		MoveL Openhole_1338, v10, fine, pHeader\WObj:=wobj0;
		MoveL Openhole_1339, v10, fine, pHeader\WObj:=wobj0;
		MoveL Openhole_1340, v10, fine, pHeader\WObj:=wobj0;
		MoveL Openhole_1341, v10, fine, pHeader\WObj:=wobj0;
		MoveL Openhole_1342, v10, fine, pHeader\WObj:=wobj0;
		MoveL Openhole_1343, v10, fine, pHeader\WObj:=wobj0;
		MoveL Openhole_1344, v10, fine, pHeader\WObj:=wobj0;
